LIN {X 0,Y 208.481,Z 945.094,A -85,B 0,C 180,E1 25559.989,E2 25559.989} C_VEL
LIN {X 0,Y 208.561,Z 942.719,A -85,B 0,C 180,E1 25564.152,E2 25564.152} C_VEL
LIN {X 0,Y 203.616,Z 945.932,A -85,B 0,C 180,E1 25571.784,E2 25571.784} C_VEL
LIN {X 0,Y 202.309,Z 947.285,A -85,B 0,C 180,E1 25573.38,E2 25573.38} C_VEL
LIN {X 0,Y 199.131,Z 950.146,A -85,B 0,C 180,E1 25574.216,E2 25574.216} C_VEL
LIN {X 0,Y 170.283,Z 972.979,A -85,B 0,C 180,E1 25579.15,E2 25579.15} C_VEL
LIN {X 0,Y 139.935,Z 991.586,A -85,B 0,C 180,E1 25586.801,E2 25586.801} C_VEL
LIN {X 0,Y 111.609,Z 1004.959,A -85,B 0,C 180,E1 25598.741,E2 25598.741} C_VEL
LIN {X 0,Y 89.534,Z 1013.124,A -85,B 0,C 180,E1 25617.669,E2 25617.669} C_VEL
LIN {X 0,Y 80.233,Z 1016.11,A -85,B 0,C 180,E1 25639.124,E2 25639.124} C_VEL
LIN {X 0,Y 80.25,Z 1016.086,A -85,B 0,C 180,E1 25660.875,E2 25660.875} C_VEL
LIN {X 0,Y 95.67,Z 1010.987,A -85,B 0,C 180,E1 25689.273,E2 25689.273} C_VEL
LIN {X 0,Y 122.761,Z 1000.055,A -85,B 0,C 180,E1 25706.77,E2 25706.77} C_VEL
LIN {X 0,Y 152.69,Z 984.282,A -85,B 0,C 180,E1 25716.747,E2 25716.747} C_VEL
LIN {X 0,Y 184.293,Z 962.437,A -85,B 0,C 180,E1 25723.376,E2 25723.376} C_VEL
LIN {X 0,Y 191.521,Z 956.574,A -85,B 0,C 180,E1 25724.562,E2 25724.562} C_VEL
LIN {X 0,Y 196.197,Z 952.595,A -85,B 0,C 180,E1 25726.225,E2 25726.225} C_VEL
LIN {X 0,Y 199.352,Z 949.805,A -85,B 0,C 180,E1 25729.978,E2 25729.978} C_VEL
LIN {X 0,Y 201.389,Z 948.643,A -85,B 0,C 180,E1 25734.136,E2 25734.136} C_VEL
LIN {X 0,Y 202.552,Z 948.131,A -85,B 0,C 180,E1 25735.725,E2 25735.725} C_VEL
LIN {X 0,Y 202.66,Z 949.809,A -85,B 0,C 180,E1 25739.218,E2 25739.218} C_VEL
LIN {X 0,Y 170.919,Z 977.867,A -85,B 0,C 180,E1 25743.237,E2 25743.237} C_VEL
LIN {X 0,Y 136.439,Z 1002.048,A -85,B 0,C 180,E1 25749.996,E2 25749.996} C_VEL
LIN {X 0,Y 103.347,Z 1020.966,A -85,B 0,C 180,E1 25762.119,E2 25762.119} C_VEL
LIN {X 0,Y 78.07,Z 1033.952,A -85,B 0,C 180,E1 25783.511,E2 25783.511} C_VEL
LIN {X 0,Y 69.524,Z 1039.389,A -85,B 0,C 180,E1 25804.18,E2 25804.18} C_VEL
LIN {X 0,Y 69.25,Z 1042.157,A -85,B 0,C 180,E1 25829.999,E2 25829.999} C_VEL
LIN {X 0,Y 69.527,Z 1039.414,A -85,B 0,C 180,E1 25855.817,E2 25855.817} C_VEL
LIN {X 0,Y 84.225,Z 1030.826,A -85,B 0,C 180,E1 25883.987,E2 25883.987} C_VEL
LIN {X 0,Y 114.045,Z 1015.315,A -85,B 0,C 180,E1 25902.786,E2 25902.786} C_VEL
LIN {X 0,Y 148.793,Z 994.172,A -85,B 0,C 180,E1 25912.78,E2 25912.78} C_VEL
LIN {X 0,Y 181.759,Z 969.208,A -85,B 0,C 180,E1 25918.286,E2 25918.286} C_VEL
LIN {X 0,Y 202.744,Z 949.964,A -85,B 0,C 180,E1 25920.772,E2 25920.772} C_VEL
LIN {X 0,Y 202.608,Z 948.314,A -85,B 0,C 180,E1 25924.274,E2 25924.274} C_VEL
LIN {X 0,Y 198.102,Z 950.964,A -85,B 0,C 180,E1 25931,E2 25931} C_VEL
LIN {X 0,Y 196.097,Z 952.662,A -85,B 0,C 180,E1 25932.195,E2 25932.195} C_VEL
LIN {X 0,Y 166.195,Z 975.484,A -85,B 0,C 180,E1 25936.959,E2 25936.959} C_VEL
LIN {X 0,Y 136.428,Z 993.025,A -85,B 0,C 180,E1 25943.915,E2 25943.915} C_VEL
LIN {X 0,Y 106.882,Z 1006.314,A -85,B 0,C 180,E1 25955.464,E2 25955.464} C_VEL
LIN {X 0,Y 85.596,Z 1013.77,A -85,B 0,C 180,E1 25971.753,E2 25971.753} C_VEL
LIN {X 0,Y 72.588,Z 1017.461,A -85,B 0,C 180,E1 25997.962,E2 25997.962} C_VEL
LIN {X 0,Y 71.763,Z 1017.732,A -85,B 0,C 180,E1 26010.001,E2 26010.001} C_VEL
LIN {X 0,Y 76.046,Z 1016.46,A -85,B 0,C 180,E1 26033.465,E2 26033.465} C_VEL
LIN {X 0,Y 94.294,Z 1010.865,A -85,B 0,C 180,E1 26056.264,E2 26056.264} C_VEL
LIN {X 0,Y 121.226,Z 1000.274,A -85,B 0,C 180,E1 26070.955,E2 26070.955} C_VEL
LIN {X 0,Y 152.847,Z 983.799,A -85,B 0,C 180,E1 26080.221,E2 26080.221} C_VEL
LIN {X 0,Y 184.689,Z 961.877,A -85,B 0,C 180,E1 26086.112,E2 26086.112} C_VEL
LIN {X 0,Y 196.094,Z 952.434,A -85,B 0,C 180,E1 26087.749,E2 26087.749} C_VEL
LIN {X 0,Y 198.088,Z 950.746,A -85,B 0,C 180,E1 26088.999,E2 26088.999} C_VEL
LIN {X 0,Y 201.389,Z 948.643,A -85,B 0,C 180,E1 26094.136,E2 26094.136} C_VEL
LIN {X 0,Y 200.229,Z 950.371,A -85,B 0,C 180,E1 26095.822,E2 26095.822} C_VEL
LIN {X 0,Y 195.34,Z 955.454,A -85,B 0,C 180,E1 26097.311,E2 26097.311} C_VEL
LIN {X 0,Y 188.146,Z 962.065,A -85,B 0,C 180,E1 26098.362,E2 26098.362} C_VEL
LIN {X 0,Y 153.922,Z 988.562,A -85,B 0,C 180,E1 26102.846,E2 26102.846} C_VEL
LIN {X 0,Y 118.999,Z 1009.936,A -85,B 0,C 180,E1 26110.728,E2 26110.728} C_VEL
LIN {X 0,Y 87.096,Z 1025.846,A -85,B 0,C 180,E1 26125.16,E2 26125.16} C_VEL
LIN {X 0,Y 67.103,Z 1035.132,A -85,B 0,C 180,E1 26147.399,E2 26147.399} C_VEL
LIN {X 0,Y 60.349,Z 1039.863,A -85,B 0,C 180,E1 26175.47,E2 26175.47} C_VEL
LIN {X 0,Y 61.337,Z 1040.787,A -85,B 0,C 180,E1 26189.999,E2 26189.999} C_VEL
LIN {X 0,Y 62.268,Z 1037.997,A -85,B 0,C 180,E1 26219.095,E2 26219.095} C_VEL
LIN {X 0,Y 79.564,Z 1029.365,A -85,B 0,C 180,E1 26248.901,E2 26248.901} C_VEL
LIN {X 0,Y 111.658,Z 1013.924,A -85,B 0,C 180,E1 26266.888,E2 26266.888} C_VEL
LIN {X 0,Y 146.132,Z 993.898,A -85,B 0,C 180,E1 26275.699,E2 26275.699} C_VEL
LIN {X 0,Y 179.53,Z 969.516,A -85,B 0,C 180,E1 26280.687,E2 26280.687} C_VEL
LIN {X 0,Y 197.003,Z 954.289,A -85,B 0,C 180,E1 26282.488,E2 26282.488} C_VEL
LIN {X 0,Y 196.533,Z 953.833,A -85,B 0,C 180,E1 26284.406,E2 26284.406} C_VEL
LIN {X 0,Y 192.985,Z 955.536,A -85,B 0,C 180,E1 26289.494,E2 26289.494} C_VEL
LIN {X 0,Y 191.197,Z 956.979,A -85,B 0,C 180,E1 26290.4,E2 26290.4} C_VEL
LIN {X 0,Y 158.897,Z 980.258,A -85,B 0,C 180,E1 26295.266,E2 26295.266} C_VEL
LIN {X 0,Y 127.117,Z 997.521,A -85,B 0,C 180,E1 26302.626,E2 26302.626} C_VEL
LIN {X 0,Y 94.244,Z 1010.583,A -85,B 0,C 180,E1 26316.562,E2 26316.562} C_VEL
LIN {X 0,Y 74.594,Z 1016.422,A -85,B 0,C 180,E1 26334.219,E2 26334.219} C_VEL
LIN {X 0,Y 63.996,Z 1019.077,A -85,B 0,C 180,E1 26370.001,E2 26370.001} C_VEL
LIN {X 0,Y 74.98,Z 1016.276,A -85,B 0,C 180,E1 26406.188,E2 26406.188} C_VEL
LIN {X 0,Y 99.778,Z 1008.6,A -85,B 0,C 180,E1 26426.569,E2 26426.569} C_VEL
LIN {X 0,Y 130.415,Z 995.771,A -85,B 0,C 180,E1 26438.238,E2 26438.238} C_VEL
LIN {X 0,Y 162.406,Z 977.795,A -85,B 0,C 180,E1 26445.282,E2 26445.282} C_VEL
LIN {X 0,Y 191.22,Z 956.727,A -85,B 0,C 180,E1 26449.567,E2 26449.567} C_VEL
LIN {X 0,Y 193.337,Z 955.08,A -85,B 0,C 180,E1 26451.002,E2 26451.002} C_VEL
LIN {X 0,Y 196.513,Z 953.635,A -85,B 0,C 180,E1 26455.593,E2 26455.593} C_VEL
LIN {X 0,Y 196.99,Z 953.973,A -85,B 0,C 180,E1 26457.275,E2 26457.275} C_VEL
LIN {X 0,Y 188.146,Z 962.065,A -85,B 0,C 180,E1 26458.362,E2 26458.362} C_VEL
LIN {X 0,Y 174.299,Z 972.838,A -85,B 0,C 180,E1 26458.579,E2 26458.579} C_VEL
LIN {X 0,Y 159.892,Z 982.792,A -85,B 0,C 180,E1 26458.877,E2 26458.877} C_VEL
LIN {X 0,Y 124.729,Z 1004.643,A -85,B 0,C 180,E1 26464.941,E2 26464.941} C_VEL
LIN {X 0,Y 90.673,Z 1021.379,A -85,B 0,C 180,E1 26476.238,E2 26476.238} C_VEL
LIN {X 0,Y 63.969,Z 1032.548,A -85,B 0,C 180,E1 26497.857,E2 26497.857} C_VEL
LIN {X 0,Y 55.242,Z 1036.551,A -85,B 0,C 180,E1 26516.76,E2 26516.76} C_VEL
LIN {X 0,Y 53.421,Z 1039.416,A -85,B 0,C 180,E1 26549.999,E2 26549.999} C_VEL
LIN {X 0,Y 55.996,Z 1036.167,A -85,B 0,C 180,E1 26585.732,E2 26585.732} C_VEL
LIN {X 0,Y 77.603,Z 1027.018,A -85,B 0,C 180,E1 26615.958,E2 26615.958} C_VEL
LIN {X 0,Y 110.855,Z 1012.045,A -85,B 0,C 180,E1 26631.405,E2 26631.405} C_VEL
LIN {X 0,Y 147.623,Z 991.18,A -85,B 0,C 180,E1 26639.34,E2 26639.34} C_VEL
LIN {X 0,Y 182.03,Z 966.196,A -85,B 0,C 180,E1 26643.568,E2 26643.568} C_VEL
LIN {X 0,Y 190.255,Z 959.17,A -85,B 0,C 180,E1 26644.552,E2 26644.552} C_VEL
LIN {X 0,Y 188.055,Z 960.104,A -85,B 0,C 180,E1 26647.598,E2 26647.598} C_VEL
LIN {X 0,Y 186.21,Z 961.356,A -85,B 0,C 180,E1 26648.52,E2 26648.52} C_VEL
LIN {X 0,Y 153.497,Z 983.679,A -85,B 0,C 180,E1 26653.094,E2 26653.094} C_VEL
LIN {X 0,Y 120.978,Z 1000.302,A -85,B 0,C 180,E1 26660.185,E2 26660.185} C_VEL
LIN {X 0,Y 89.81,Z 1011.934,A -85,B 0,C 180,E1 26672.555,E2 26672.555} C_VEL
LIN {X 0,Y 69.429,Z 1017.52,A -85,B 0,C 180,E1 26689.143,E2 26689.143} C_VEL
LIN {X 0,Y 57.436,Z 1020.161,A -85,B 0,C 180,E1 26714.717,E2 26714.717} C_VEL
LIN {X 0,Y 56.215,Z 1020.425,A -85,B 0,C 180,E1 26730.001,E2 26730.001} C_VEL
LIN {X 0,Y 62.04,Z 1019.166,A -85,B 0,C 180,E1 26759.215,E2 26759.215} C_VEL
LIN {X 0,Y 84.258,Z 1013.575,A -85,B 0,C 180,E1 26783.959,E2 26783.959} C_VEL
LIN {X 0,Y 114.463,Z 1002.997,A -85,B 0,C 180,E1 26797.804,E2 26797.804} C_VEL
LIN {X 0,Y 148.299,Z 986.544,A -85,B 0,C 180,E1 26805.898,E2 26805.898} C_VEL
LIN {X 0,Y 181.094,Z 965.062,A -85,B 0,C 180,E1 26810.817,E2 26810.817} C_VEL
LIN {X 0,Y 186.185,Z 961.16,A -85,B 0,C 180,E1 26811.424,E2 26811.424} C_VEL
LIN {X 0,Y 188.053,Z 959.89,A -85,B 0,C 180,E1 26812.363,E2 26812.363} C_VEL
LIN {X 0,Y 190.247,Z 958.961,A -85,B 0,C 180,E1 26815.448,E2 26815.448} C_VEL
LIN {X 0,Y 159.892,Z 982.792,A -85,B 0,C 180,E1 26818.877,E2 26818.877} C_VEL
LIN {X 0,Y 144.954,Z 992.033,A -85,B 0,C 180,E1 26819.311,E2 26819.311} C_VEL
LIN {X 0,Y 129.62,Z 1000.319,A -85,B 0,C 180,E1 26820.051,E2 26820.051} C_VEL
LIN {X 0,Y 92.14,Z 1018.502,A -85,B 0,C 180,E1 26829.635,E2 26829.635} C_VEL
LIN {X 0,Y 60.304,Z 1030.74,A -85,B 0,C 180,E1 26850.181,E2 26850.181} C_VEL
LIN {X 0,Y 48.583,Z 1035.127,A -85,B 0,C 180,E1 26871.443,E2 26871.443} C_VEL
LIN {X 0,Y 45.456,Z 1038.036,A -85,B 0,C 180,E1 26910.215,E2 26910.215} C_VEL
LIN {X 0,Y 48.588,Z 1035.156,A -85,B 0,C 180,E1 26948.548,E2 26948.548} C_VEL
LIN {X 0,Y 74.079,Z 1025.748,A -85,B 0,C 180,E1 26981.571,E2 26981.571} C_VEL
LIN {X 0,Y 109.912,Z 1010.576,A -85,B 0,C 180,E1 26995.753,E2 26995.753} C_VEL
LIN {X 0,Y 147.708,Z 989.735,A -85,B 0,C 180,E1 27002.61,E2 27002.61} C_VEL
LIN {X 0,Y 181.435,Z 965.747,A -85,B 0,C 180,E1 27006.083,E2 27006.083} C_VEL
LIN {X 0,Y 178.5,Z 967.827,A -85,B 0,C 180,E1 27006.865,E2 27006.865} C_VEL
LIN {X 0,Y 142.994,Z 990.031,A -85,B 0,C 180,E1 27011.661,E2 27011.661} C_VEL
LIN {X 0,Y 108.313,Z 1005.767,A -85,B 0,C 180,E1 27019.352,E2 27019.352} C_VEL
LIN {X 0,Y 74.136,Z 1016.459,A -85,B 0,C 180,E1 27035.229,E2 27035.229} C_VEL
LIN {X 0,Y 55.339,Z 1020.551,A -85,B 0,C 180,E1 27056.829,E2 27056.829} C_VEL
LIN {X 0,Y 48.447,Z 1021.771,A -85,B 0,C 180,E1 27090.001,E2 27090.001} C_VEL
LIN {X 0,Y 60.401,Z 1019.589,A -85,B 0,C 180,E1 27131.301,E2 27131.301} C_VEL
LIN {X 0,Y 92.087,Z 1011.312,A -85,B 0,C 180,E1 27154.723,E2 27154.723} C_VEL
LIN {X 0,Y 125.467,Z 998.495,A -85,B 0,C 180,E1 27164.874,E2 27164.874} C_VEL
LIN {X 0,Y 159.161,Z 980.563,A -85,B 0,C 180,E1 27170.719,E2 27170.719} C_VEL
LIN {X 0,Y 178.711,Z 967.456,A -85,B 0,C 180,E1 27173.117,E2 27173.117} C_VEL
LIN {X 0,Y 181.498,Z 965.489,A -85,B 0,C 180,E1 27173.885,E2 27173.885} C_VEL
LIN {X 0,Y 145.617,Z 990.907,A -85,B 0,C 180,E1 27177.625,E2 27177.625} C_VEL
LIN {X 0,Y 129.62,Z 1000.319,A -85,B 0,C 180,E1 27180.051,E2 27180.051} C_VEL
LIN {X 0,Y 113.806,Z 1007.736,A -85,B 0,C 180,E1 27181.081,E2 27181.081} C_VEL
LIN {X 0,Y 97.76,Z 1014.25,A -85,B 0,C 180,E1 27182.495,E2 27182.495} C_VEL
LIN {X 0,Y 63.393,Z 1027.055,A -85,B 0,C 180,E1 27197.191,E2 27197.191} C_VEL
LIN {X 0,Y 41.606,Z 1034.004,A -85,B 0,C 180,E1 27226.775,E2 27226.775} C_VEL
LIN {X 0,Y 37.539,Z 1036.664,A -85,B 0,C 180,E1 27269.998,E2 27269.998} C_VEL
LIN {X 0,Y 42.435,Z 1033.724,A -85,B 0,C 180,E1 27315.523,E2 27315.523} C_VEL
LIN {X 0,Y 71.4,Z 1024.45,A -85,B 0,C 180,E1 27347.727,E2 27347.727} C_VEL
LIN {X 0,Y 111.203,Z 1008.342,A -85,B 0,C 180,E1 27360.515,E2 27360.515} C_VEL
LIN {X 0,Y 149.532,Z 987.498,A -85,B 0,C 180,E1 27366.022,E2 27366.022} C_VEL
LIN {X 0,Y 155.275,Z 983.914,A -85,B 0,C 180,E1 27366.579,E2 27366.579} C_VEL
LIN {X 0,Y 120.064,Z 1001.594,A -85,B 0,C 180,E1 27372.245,E2 27372.245} C_VEL
LIN {X 0,Y 88.554,Z 1012.908,A -85,B 0,C 180,E1 27380.805,E2 27380.805} C_VEL
LIN {X 0,Y 58.517,Z 1020.225,A -85,B 0,C 180,E1 27399.089,E2 27399.089} C_VEL
LIN {X 0,Y 42.597,Z 1022.861,A -85,B 0,C 180,E1 27429.182,E2 27429.182} C_VEL
LIN {X 0,Y 40.666,Z 1023.118,A -85,B 0,C 180,E1 27450.001,E2 27450.001} C_VEL
LIN {X 0,Y 49.031,Z 1021.864,A -85,B 0,C 180,E1 27488.14,E2 27488.14} C_VEL
LIN {X 0,Y 76.12,Z 1016.285,A -85,B 0,C 180,E1 27513.514,E2 27513.514} C_VEL
LIN {X 0,Y 109.521,Z 1005.72,A -85,B 0,C 180,E1 27525.392,E2 27525.392} C_VEL
LIN {X 0,Y 145.149,Z 989.377,A -85,B 0,C 180,E1 27531.858,E2 27531.858} C_VEL
LIN {X 0,Y 155.572,Z 983.551,A -85,B 0,C 180,E1 27533.371,E2 27533.371} C_VEL
LIN {X 0,Y 117.838,Z 1005.099,A -85,B 0,C 180,E1 27538.229,E2 27538.229} C_VEL
LIN {X 0,Y 97.76,Z 1014.25,A -85,B 0,C 180,E1 27542.495,E2 27542.495} C_VEL
LIN {X 0,Y 81.484,Z 1019.912,A -85,B 0,C 180,E1 27544.592,E2 27544.592} C_VEL
LIN {X 0,Y 65.026,Z 1024.534,A -85,B 0,C 180,E1 27547.795,E2 27547.795} C_VEL
LIN {X 0,Y 37.104,Z 1032.259,A -85,B 0,C 180,E1 27575.303,E2 27575.303} C_VEL
LIN {X 0,Y 29.543,Z 1035.28,A -85,B 0,C 180,E1 27629.998,E2 27629.998} C_VEL
LIN {X 0,Y 37.104,Z 1032.288,A -85,B 0,C 180,E1 27684.692,E2 27684.692} C_VEL
LIN {X 0,Y 70.091,Z 1022.984,A -85,B 0,C 180,E1 27714.495,E2 27714.495} C_VEL
LIN {X 0,Y 111.495,Z 1006.919,A -85,B 0,C 180,E1 27724.858,E2 27724.858} C_VEL
LIN {X 0,Y 126.179,Z 999.786,A -85,B 0,C 180,E1 27726.873,E2 27726.873} C_VEL
LIN {X 0,Y 111.394,Z 1005.798,A -85,B 0,C 180,E1 27729.817,E2 27729.817} C_VEL
LIN {X 0,Y 79.67,Z 1016.006,A -85,B 0,C 180,E1 27738.168,E2 27738.168} C_VEL
LIN {X 0,Y 46.159,Z 1022.815,A -85,B 0,C 180,E1 27760.926,E2 27760.926} C_VEL
LIN {X 0,Y 32.897,Z 1024.464,A -85,B 0,C 180,E1 27810.002,E2 27810.002} C_VEL
LIN {X 0,Y 46.448,Z 1022.741,A -85,B 0,C 180,E1 27859.383,E2 27859.383} C_VEL
LIN {X 0,Y 79.703,Z 1015.923,A -85,B 0,C 180,E1 27881.765,E2 27881.765} C_VEL
LIN {X 0,Y 118.679,Z 1002.82,A -85,B 0,C 180,E1 27891.37,E2 27891.37} C_VEL
LIN {X 0,Y 126.095,Z 999.712,A -85,B 0,C 180,E1 27893.123,E2 27893.123} C_VEL
LIN {X 0,Y 86.928,Z 1017.032,A -85,B 0,C 180,E1 27900.026,E2 27900.026} C_VEL
LIN {X 0,Y 65.026,Z 1024.534,A -85,B 0,C 180,E1 27907.795,E2 27907.795} C_VEL
LIN {X 0,Y 48.765,Z 1028.181,A -85,B 0,C 180,E1 27913.264,E2 27913.264} C_VEL
LIN {X 0,Y 32.912,Z 1030.836,A -85,B 0,C 180,E1 27923.579,E2 27923.579} C_VEL
LIN {X 0,Y 21.549,Z 1033.895,A -85,B 0,C 180,E1 27989.997,E2 27989.997} C_VEL
LIN {X 0,Y 33.003,Z 1030.848,A -85,B 0,C 180,E1 28056.558,E2 28056.558} C_VEL
LIN {X 0,Y 70.1,Z 1021.426,A -85,B 0,C 180,E1 28081.494,E2 28081.494} C_VEL
LIN {X 0,Y 97.391,Z 1011.851,A -85,B 0,C 180,E1 28087.202,E2 28087.202} C_VEL
LIN {X 0,Y 82.822,Z 1016.043,A -85,B 0,C 180,E1 28091.179,E2 28091.179} C_VEL
LIN {X 0,Y 50.158,Z 1022.93,A -85,B 0,C 180,E1 28105.109,E2 28105.109} C_VEL
LIN {X 0,Y 28.568,Z 1025.562,A -85,B 0,C 180,E1 28138,E2 28138} C_VEL
LIN {X 0,Y 25.103,Z 1025.814,A -85,B 0,C 180,E1 28170.002,E2 28170.002} C_VEL
LIN {X 0,Y 37.994,Z 1024.57,A -85,B 0,C 180,E1 28222.843,E2 28222.843} C_VEL
LIN {X 0,Y 70.542,Z 1019.003,A -85,B 0,C 180,E1 28244.974,E2 28244.974} C_VEL
LIN {X 0,Y 92.006,Z 1013.302,A -85,B 0,C 180,E1 28250.872,E2 28250.872} C_VEL
LIN {X 0,Y 97.531,Z 1011.701,A -85,B 0,C 180,E1 28252.757,E2 28252.757} C_VEL
LIN {X 0,Y 56.874,Z 1025.178,A -85,B 0,C 180,E1 28263.362,E2 28263.362} C_VEL
LIN {X 0,Y 32.912,Z 1030.836,A -85,B 0,C 180,E1 28283.579,E2 28283.579} C_VEL
LIN {X 0,Y 22.965,Z 1032.258,A -85,B 0,C 180,E1 28301.464,E2 28301.464} C_VEL
LIN {X 0,Y 14.696,Z 1032.569,A -85,B 0,C 180,E1 28334.454,E2 28334.454} C_VEL
LIN {X 0,Y 13.198,Z 1032.165,A -85,B 0,C 180,E1 28371.239,E2 28371.239} C_VEL
LIN {X 0,Y 36.928,Z 1028.247,A -85,B 0,C 180,E1 28436.174,E2 28436.174} C_VEL
LIN {X 0,Y 69.266,Z 1020.44,A -85,B 0,C 180,E1 28448.058,E2 28448.058} C_VEL
LIN {X 0,Y 47.373,Z 1024.284,A -85,B 0,C 180,E1 28456.516,E2 28456.516} C_VEL
LIN {X 0,Y 22.35,Z 1026.91,A -85,B 0,C 180,E1 28487.362,E2 28487.362} C_VEL
LIN {X 0,Y 17.333,Z 1027.16,A -85,B 0,C 180,E1 28530.004,E2 28530.004} C_VEL
LIN {X 0,Y 34.174,Z 1025.888,A -85,B 0,C 180,E1 28593.779,E2 28593.779} C_VEL
LIN {X 0,Y 61.66,Z 1021.808,A -85,B 0,C 180,E1 28609.166,E2 28609.166} C_VEL
LIN {X 0,Y 69.284,Z 1020.373,A -85,B 0,C 180,E1 28611.942,E2 28611.942} C_VEL
LIN {X 0,Y 28.124,Z 1029.799,A -85,B 0,C 180,E1 28631.81,E2 28631.81} C_VEL
LIN {X 0,Y 13.522,Z 1032.505,A -85,B 0,C 180,E1 28709.995,E2 28709.995} C_VEL
LIN {X 0,Y 13.198,Z 1032.165,A -85,B 0,C 180,E1 28731.239,E2 28731.239} C_VEL
LIN {X 0,Y 17.713,Z 1030.8,A -85,B 0,C 180,E1 28778.396,E2 28778.396} C_VEL
LIN {X 0,Y 35.288,Z 1027.148,A -85,B 0,C 180,E1 28808.439,E2 28808.439} C_VEL
LIN {X 0,Y 31.153,Z 1027.306,A -85,B 0,C 180,E1 28813.603,E2 28813.603} C_VEL
LIN {X 0,Y 9.538,Z 1028.51,A -85,B 0,C 180,E1 28890.006,E2 28890.006} C_VEL
LIN {X 0,Y 31.16,Z 1027.274,A -85,B 0,C 180,E1 28966.357,E2 28966.357} C_VEL
LIN {X 0,Y 35.96,Z 1027.005,A -85,B 0,C 180,E1 28971.339,E2 28971.339} C_VEL
LIN {X 0,Y 15.213,Z 1029.998,A -85,B 0,C 180,E1 28985.589,E2 28985.589} C_VEL
LIN {X 0,Y 5.49,Z 1031.113,A -85,B 0,C 180,E1 29069.989,E2 29069.989} C_VEL
LIN {X 0,Y 30.478,Z 1027.973,A -85,B 0,C 180,E1 29166.556,E2 29166.556} C_VEL
LIN {X 0,Y 35.288,Z 1027.148,A -85,B 0,C 180,E1 29168.439,E2 29168.439} C_VEL
LIN {X 0,Y 37.572,Z 1029.121,A -85,B 0,C 180,E1 29169.161,E2 29169.161} C_VEL
LIN {X 0,Y 37.572,Z 1104,A -85,B 0,C 180,E1 29169.161,E2 29169.161} C_VEL
LIN {X 0,Y 37.572,Z 1104,A -85,B 0,C 180,E1 29169.161,E2 29169.161}

QRS_NEXT_CUT()
PTP {E1 29337.043,E2 29337.043}
PTP {X 0,Y 607.835,A -85,B 0,C 180,E1 29337.043,E2 29337.043,E3 0,E4 0,E5 0,E6 0}
QRS_SPEED_INIT()
LIN {X 0,Y 607.835,Z 1104,A -85,B 0,C 180,E1 29337.043,E2 29337.043,E3 0,E4 0,E5 0,E6 0} C_VEL
LIN {X 0,Y 607.835,Z 381.402,A -85,B 0,C 180,E1 29337.043,E2 29337.043} C_VEL
LIN {X 0,Y 607.835,Z 373.326,A -85,B 0,C 180,E1 29337.043,E2 29337.043} C_VEL
LIN {X 0,Y 607.835,Z 371.326,A -85,B 0,C 180,E1 29336.855,E2 29336.855} C_VEL
LIN {X 0,Y 607.918,Z 371.324,A -85,B 0,C 180,E1 29333.768,E2 29333.768} C_VEL
LIN {X 0,Y 607.836,Z 371.325,A -85,B 0,C 180,E1 29330.723,E2 29330.723} C_VEL
LIN {X 0,Y 607.886,Z 371.327,A -85,B 0,C 180,E1 29327.846,E2 29327.846} C_VEL
LIN {X 0,Y 607.847,Z 371.324,A -85,B 0,C 180,E1 29324.74,E2 29324.74} C_VEL
LIN {X 0,Y 607.849,Z 371.326,A -85,B 0,C 180,E1 29321.946,E2 29321.946} C_VEL
LIN {X 0,Y 607.866,Z 371.324,A -85,B 0,C 180,E1 29318.683,E2 29318.683} C_VEL
LIN {X 0,Y 607.838,Z 371.326,A -85,B 0,C 180,E1 29315.916,E2 29315.916} C_VEL
LIN {X 0,Y 607.919,Z 371.324,A -85,B 0,C 180,E1 29312.849,E2 29312.849} C_VEL
LIN {X 0,Y 607.839,Z 371.324,A -85,B 0,C 180,E1 29309.778,E2 29309.778} C_VEL
LIN {X 0,Y 607.908,Z 371.328,A -85,B 0,C 180,E1 29306.79,E2 29306.79} C_VEL
LIN {X 0,Y 607.844,Z 371.323,A -85,B 0,C 180,E1 29303.688,E2 29303.688} C_VEL
LIN {X 0,Y 607.871,Z 371.327,A -85,B 0,C 180,E1 29300.83,E2 29300.83} C_VEL
LIN {X 0,Y 607.854,Z 371.324,A -85,B 0,C 180,E1 29297.591,E2 29297.591} C_VEL
LIN {X 0,Y 607.848,Z 371.325,A -85,B 0,C 180,E1 29294.849,E2 29294.849} C_VEL
LIN {X 0,Y 607.894,Z 371.322,A -85,B 0,C 180,E1 29291.691,E2 29291.691} C_VEL
LIN {X 0,Y 607.843,Z 371.326,A -85,B 0,C 180,E1 29288.767,E2 29288.767} C_VEL
LIN {X 0,Y 607.917,Z 371.325,A -85,B 0,C 180,E1 29285.724,E2 29285.724} C_VEL
LIN {X 0,Y 607.889,Z 371.537,A -85,B 0,C 180,E1 29283.975,E2 29283.975} C_VEL
LIN {X 0,Y 607.908,Z 373.819,A -85,B 0,C 180,E1 29283.775,E2 29283.775} C_VEL
LIN {X 0,Y 607.876,Z 417.731,A -85,B 0,C 180,E1 29280.932,E2 29280.932} C_VEL
LIN {X 0,Y 607.895,Z 463.368,A -85,B 0,C 180,E1 29278.061,E2 29278.061} C_VEL
LIN {X 0,Y 607.889,Z 470.207,A -85,B 0,C 180,E1 29277.648,E2 29277.648} C_VEL
LIN {X 0,Y 607.906,Z 714.954,A -85,B 0,C 180,E1 29274.487,E2 29274.487} C_VEL
LIN {X 0,Y 607.916,Z 737.553,A -85,B 0,C 180,E1 29274.138,E2 29274.138} C_VEL
LIN {X 0,Y 607.905,Z 756.795,A -85,B 0,C 180,E1 29273.687,E2 29273.687} C_VEL
LIN {X 0,Y 607.915,Z 776.617,A -85,B 0,C 180,E1 29273.045,E2 29273.045} C_VEL
LIN {X 0,Y 607.906,Z 794.968,A -85,B 0,C 180,E1 29272.279,E2 29272.279} C_VEL
LIN {X 0,Y 607.918,Z 813.819,A -85,B 0,C 180,E1 29271.315,E2 29271.315} C_VEL
LIN {X 0,Y 607.917,Z 831.797,A -85,B 0,C 180,E1 29270.206,E2 29270.206} C_VEL
LIN {X 0,Y 607.916,Z 848.757,A -85,B 0,C 180,E1 29268.964,E2 29268.964} C_VEL
LIN {X 0,Y 607.916,Z 864.943,A -85,B 0,C 180,E1 29267.566,E2 29267.566} C_VEL
LIN {X 0,Y 607.909,Z 879.945,A -85,B 0,C 180,E1 29266.041,E2 29266.041} C_VEL
LIN {X 0,Y 607.915,Z 893.927,A -85,B 0,C 180,E1 29264.361,E2 29264.361} C_VEL
LIN {X 0,Y 607.917,Z 905.994,A -85,B 0,C 180,E1 29262.636,E2 29262.636} C_VEL
LIN {X 0,Y 607.907,Z 916.116,A -85,B 0,C 180,E1 29260.903,E2 29260.903} C_VEL
LIN {X 0,Y 607.901,Z 924.868,A -85,B 0,C 180,E1 29259.085,E2 29259.085} C_VEL
LIN {X 0,Y 607.9,Z 931.847,A -85,B 0,C 180,E1 29257.276,E2 29257.276} C_VEL
LIN {X 0,Y 607.901,Z 937.387,A -85,B 0,C 180,E1 29255.38,E2 29255.38} C_VEL
LIN {X 0,Y 607.9,Z 941.164,A -85,B 0,C 180,E1 29253.489,E2 29253.489} C_VEL
LIN {X 0,Y 607.903,Z 943.341,A -85,B 0,C 180,E1 29251.602,E2 29251.602} C_VEL
LIN {X 0,Y 607.904,Z 943.95,A -85,B 0,C 180,E1 29249.717,E2 29249.717} C_VEL
LIN {X 0,Y 607.915,Z 942.998,A -85,B 0,C 180,E1 29247.832,E2 29247.832} C_VEL
LIN {X 0,Y 607.917,Z 940.209,A -85,B 0,C 180,E1 29245.85,E2 29245.85} C_VEL
LIN {X 0,Y 607.915,Z 935.855,A -85,B 0,C 180,E1 29243.958,E2 29243.958} C_VEL
LIN {X 0,Y 607.91,Z 929.786,A -85,B 0,C 180,E1 29242.059,E2 29242.059} C_VEL
LIN {X 0,Y 607.905,Z 922.315,A -85,B 0,C 180,E1 29240.246,E2 29240.246} C_VEL
LIN {X 0,Y 607.904,Z 912.972,A -85,B 0,C 180,E1 29238.424,E2 29238.424} C_VEL
LIN {X 0,Y 607.906,Z 902.111,A -85,B 0,C 180,E1 29236.687,E2 29236.687} C_VEL
LIN {X 0,Y 607.914,Z 889.841,A -85,B 0,C 180,E1 29235.035,E2 29235.035} C_VEL
LIN {X 0,Y 607.917,Z 876.164,A -85,B 0,C 180,E1 29233.469,E2 29233.469} C_VEL
LIN {X 0,Y 607.912,Z 861,A -85,B 0,C 180,E1 29231.988,E2 29231.988} C_VEL
LIN {X 0,Y 607.918,Z 844.197,A -85,B 0,C 180,E1 29230.595,E2 29230.595} C_VEL
LIN {X 0,Y 607.917,Z 827.063,A -85,B 0,C 180,E1 29229.392,E2 29229.392} C_VEL
LIN {X 0,Y 607.918,Z 808.945,A -85,B 0,C 180,E1 29228.322,E2 29228.322} C_VEL
LIN {X 0,Y 607.914,Z 790.231,A -85,B 0,C 180,E1 29227.415,E2 29227.415} C_VEL
LIN {X 0,Y 607.917,Z 771.118,A -85,B 0,C 180,E1 29226.673,E2 29226.673} C_VEL
LIN {X 0,Y 607.906,Z 751.358,A -85,B 0,C 180,E1 29226.082,E2 29226.082} C_VEL
LIN {X 0,Y 607.913,Z 731.468,A -85,B 0,C 180,E1 29225.657,E2 29225.657} C_VEL
LIN {X 0,Y 607.883,Z 470.115,A -85,B 0,C 180,E1 29222.258,E2 29222.258} C_VEL
LIN {X 0,Y 607.878,Z 425.789,A -85,B 0,C 180,E1 29219.491,E2 29219.491} C_VEL
LIN {X 0,Y 607.917,Z 380.359,A -85,B 0,C 180,E1 29216.565,E2 29216.565} C_VEL
LIN {X 0,Y 607.895,Z 371.672,A -85,B 0,C 180,E1 29215.966,E2 29215.966} C_VEL
LIN {X 0,Y 607.851,Z 371.324,A -85,B 0,C 180,E1 29215.31,E2 29215.31} C_VEL
LIN {X 0,Y 607.919,Z 371.321,A -85,B 0,C 180,E1 29212.277,E2 29212.277} C_VEL
LIN {X 0,Y 607.852,Z 371.324,A -85,B 0,C 180,E1 29209.171,E2 29209.171} C_VEL
LIN {X 0,Y 607.9,Z 371.321,A -85,B 0,C 180,E1 29206.175,E2 29206.175} C_VEL
LIN {X 0,Y 607.857,Z 371.325,A -85,B 0,C 180,E1 29203.05,E2 29203.05} C_VEL
LIN {X 0,Y 607.871,Z 371.322,A -85,B 0,C 180,E1 29200.15,E2 29200.15} C_VEL
LIN {X 0,Y 607.864,Z 371.325,A -85,B 0,C 180,E1 29196.897,E2 29196.897} C_VEL
LIN {X 0,Y 607.859,Z 371.323,A -85,B 0,C 180,E1 29194.001,E2 29194.001} C_VEL
LIN {X 0,Y 607.864,Z 371.325,A -85,B 0,C 180,E1 29190.658,E2 29190.658} C_VEL
LIN {X 0,Y 607.85,Z 371.324,A -85,B 0,C 180,E1 29187.85,E2 29187.85} C_VEL
LIN {X 0,Y 607.898,Z 371.327,A -85,B 0,C 180,E1 29184.694,E2 29184.694} C_VEL
LIN {X 0,Y 607.844,Z 371.324,A -85,B 0,C 180,E1 29181.723,E2 29181.723} C_VEL
LIN {X 0,Y 607.914,Z 371.327,A -85,B 0,C 180,E1 29178.607,E2 29178.607} C_VEL
LIN {X 0,Y 607.842,Z 371.325,A -85,B 0,C 180,E1 29175.651,E2 29175.651} C_VEL
LIN {X 0,Y 607.893,Z 371.323,A -85,B 0,C 180,E1 29172.733,E2 29172.733} C_VEL
LIN {X 0,Y 607.846,Z 371.326,A -85,B 0,C 180,E1 29169.564,E2 29169.564} C_VEL
LIN {X 0,Y 607.854,Z 371.324,A -85,B 0,C 180,E1 29166.802,E2 29166.802} C_VEL
LIN {X 0,Y 607.858,Z 371.326,A -85,B 0,C 180,E1 29163.49,E2 29163.49} C_VEL
LIN {X 0,Y 607.841,Z 371.325,A -85,B 0,C 180,E1 29160.754,E2 29160.754} C_VEL
LIN {X 0,Y 607.909,Z 371.327,A -85,B 0,C 180,E1 29157.644,E2 29157.644} C_VEL
LIN {X 0,Y 607.836,Z 371.326,A -85,B 0,C 180,E1 29154.715,E2 29154.715} C_VEL
LIN {X 0,Y 607.896,Z 371.323,A -85,B 0,C 180,E1 29151.773,E2 29151.773} C_VEL
LIN {X 0,Y 607.839,Z 371.325,A -85,B 0,C 180,E1 29148.635,E2 29148.635} C_VEL
LIN {X 0,Y 607.849,Z 371.324,A -85,B 0,C 180,E1 29145.91,E2 29145.91} C_VEL
LIN {X 0,Y 607.85,Z 371.326,A -85,B 0,C 180,E1 29142.565,E2 29142.565} C_VEL
LIN {X 0,Y 607.838,Z 371.324,A -85,B 0,C 180,E1 29139.792,E2 29139.792} C_VEL
LIN {X 0,Y 607.889,Z 371.327,A -85,B 0,C 180,E1 29136.647,E2 29136.647} C_VEL
LIN {X 0,Y 607.831,Z 371.325,A -85,B 0,C 180,E1 29133.737,E2 29133.737} C_VEL
LIN {X 0,Y 607.914,Z 371.327,A -85,B 0,C 180,E1 29130.651,E2 29130.651} C_VEL
LIN {X 0,Y 607.832,Z 371.327,A -85,B 0,C 180,E1 29127.683,E2 29127.683} C_VEL
LIN {X 0,Y 607.847,Z 371.325,A -85,B 0,C 180,E1 29124.965,E2 29124.965} C_VEL
LIN {X 0,Y 607.845,Z 371.326,A -85,B 0,C 180,E1 29121.674,E2 29121.674} C_VEL
LIN {X 0,Y 607.829,Z 371.327,A -85,B 0,C 180,E1 29118.979,E2 29118.979} C_VEL
LIN {X 0,Y 607.91,Z 371.328,A -85,B 0,C 180,E1 29115.915,E2 29115.915} C_VEL
LIN {X 0,Y 607.825,Z 371.319,A -85,B 0,C 180,E1 29112.924,E2 29112.924} C_VEL
LIN {X 0,Y 607.883,Z 371.652,A -85,B 0,C 180,E1 29112.08,E2 29112.08} C_VEL
LIN {X 0,Y 607.904,Z 373.549,A -85,B 0,C 180,E1 29111.935,E2 29111.935} C_VEL
LIN {X 0,Y 607.918,Z 430.557,A -85,B 0,C 180,E1 29109.077,E2 29109.077} C_VEL
LIN {X 0,Y 607.904,Z 466.026,A -85,B 0,C 180,E1 29107.384,E2 29107.384} C_VEL
LIN {X 0,Y 607.915,Z 668.583,A -85,B 0,C 180,E1 29104.485,E2 29104.485} C_VEL
LIN {X 0,Y 607.913,Z 815.111,A -85,B 0,C 180,E1 29102.425,E2 29102.425} C_VEL
LIN {X 0,Y 607.914,Z 837.997,A -85,B 0,C 180,E1 29101.932,E2 29101.932} C_VEL
LIN {X 0,Y 607.918,Z 856.544,A -85,B 0,C 180,E1 29101.394,E2 29101.394} C_VEL
LIN {X 0,Y 607.912,Z 877.921,A -85,B 0,C 180,E1 29100.628,E2 29100.628} C_VEL
LIN {X 0,Y 607.919,Z 898.106,A -85,B 0,C 180,E1 29099.726,E2 29099.726} C_VEL
LIN {X 0,Y 607.916,Z 918.757,A -85,B 0,C 180,E1 29098.649,E2 29098.649} C_VEL
LIN {X 0,Y 607.918,Z 938.559,A -85,B 0,C 180,E1 29097.421,E2 29097.421} C_VEL
LIN {X 0,Y 607.912,Z 957.955,A -85,B 0,C 180,E1 29096.05,E2 29096.05} C_VEL
LIN {X 0,Y 607.91,Z 976.18,A -85,B 0,C 180,E1 29094.558,E2 29094.558} C_VEL
LIN {X 0,Y 607.909,Z 994.595,A -85,B 0,C 180,E1 29092.84,E2 29092.84} C_VEL
LIN {X 0,Y 607.916,Z 1010.874,A -85,B 0,C 180,E1 29091.112,E2 29091.112} C_VEL
LIN {X 0,Y 607.913,Z 1026.064,A -85,B 0,C 180,E1 29089.253,E2 29089.253} C_VEL
LIN {X 0,Y 607.913,Z 1040.516,A -85,B 0,C 180,E1 29087.221,E2 29087.221} C_VEL
LIN {X 0,Y 607.9,Z 1052.034,A -85,B 0,C 180,E1 29085.356,E2 29085.356} C_VEL
LIN {X 0,Y 607.885,Z 1062.754,A -85,B 0,C 180,E1 29083.313,E2 29083.313} C_VEL
LIN {X 0,Y 607.907,Z 1071.374,A -85,B 0,C 180,E1 29081.383,E2 29081.383} C_VEL
LIN {X 0,Y 607.896,Z 1079.037,A -85,B 0,C 180,E1 29079.276,E2 29079.276} C_VEL
LIN {X 0,Y 607.894,Z 1084.335,A -85,B 0,C 180,E1 29077.466,E2 29077.466} C_VEL
LIN {X 0,Y 607.908,Z 1089.161,A -85,B 0,C 180,E1 29075.285,E2 29075.285} C_VEL
LIN {X 0,Y 607.884,Z 1091.953,A -85,B 0,C 180,E1 29073.395,E2 29073.395} C_VEL
LIN {X 0,Y 607.909,Z 1093.716,A -85,B 0,C 180,E1 29071.225,E2 29071.225} C_VEL
LIN {X 0,Y 607.883,Z 1093.828,A -85,B 0,C 180,E1 29069.246,E2 29069.246} C_VEL
LIN {X 0,Y 607.895,Z 1092.63,A -85,B 0,C 180,E1 29067.172,E2 29067.172} C_VEL
LIN {X 0,Y 607.903,Z 1089.797,A -85,B 0,C 180,E1 29065.094,E2 29065.094} C_VEL
LIN {X 0,Y 607.882,Z 1085.597,A -85,B 0,C 180,E1 29063.009,E2 29063.009} C_VEL
LIN {X 0,Y 607.913,Z 1079.647,A -85,B 0,C 180,E1 29060.915,E2 29060.915} C_VEL
LIN {X 0,Y 607.897,Z 1072.187,A -85,B 0,C 180,E1 29058.809,E2 29058.809} C_VEL
LIN {X 0,Y 607.887,Z 1063.218,A -85,B 0,C 180,E1 29056.784,E2 29056.784} C_VEL
LIN {X 0,Y 607.911,Z 1053.18,A -85,B 0,C 180,E1 29054.84,E2 29054.84} C_VEL
LIN {X 0,Y 607.912,Z 1041.043,A -85,B 0,C 180,E1 29052.86,E2 29052.86} C_VEL
LIN {X 0,Y 607.912,Z 1027.214,A -85,B 0,C 180,E1 29050.895,E2 29050.895} C_VEL
LIN {X 0,Y 607.917,Z 1012.578,A -85,B 0,C 180,E1 29049.089,E2 29049.089} C_VEL
LIN {X 0,Y 607.905,Z 996.233,A -85,B 0,C 180,E1 29047.325,E2 29047.325} C_VEL
LIN {X 0,Y 607.905,Z 978.853,A -85,B 0,C 180,E1 29045.67,E2 29045.67} C_VEL
LIN {X 0,Y 607.908,Z 960.603,A -85,B 0,C 180,E1 29044.16,E2 29044.16} C_VEL
LIN {X 0,Y 607.918,Z 940.163,A -85,B 0,C 180,E1 29042.685,E2 29042.685} C_VEL
LIN {X 0,Y 607.916,Z 920.827,A -85,B 0,C 180,E1 29041.474,E2 29041.474} C_VEL
LIN {X 0,Y 607.918,Z 900.293,A -85,B 0,C 180,E1 29040.38,E2 29040.38} C_VEL
LIN {X 0,Y 607.914,Z 881.45,A -85,B 0,C 180,E1 29039.523,E2 29039.523} C_VEL
LIN {X 0,Y 607.915,Z 859.018,A -85,B 0,C 180,E1 29038.685,E2 29038.685} C_VEL
LIN {X 0,Y 607.912,Z 840.386,A -85,B 0,C 180,E1 29038.132,E2 29038.132} C_VEL
LIN {X 0,Y 607.912,Z 818.534,A -85,B 0,C 180,E1 29037.631,E2 29037.631} C_VEL
LIN {X 0,Y 607.913,Z 775.337,A -85,B 0,C 180,E1 29037.001,E2 29037.001} C_VEL
LIN {X 0,Y 607.902,Z 568.743,A -85,B 0,C 180,E1 29034.1,E2 29034.1} C_VEL
LIN {X 0,Y 607.905,Z 465.312,A -85,B 0,C 180,E1 29032.6,E2 29032.6} C_VEL
LIN {X 0,Y 607.916,Z 407.824,A -85,B 0,C 180,E1 29029.798,E2 29029.798} C_VEL
LIN {X 0,Y 607.892,Z 372.115,A -85,B 0,C 180,E1 29027.976,E2 29027.976} C_VEL
LIN {X 0,Y 607.873,Z 371.406,A -85,B 0,C 180,E1 29027.848,E2 29027.848} C_VEL
LIN {X 0,Y 607.826,Z 371.327,A -85,B 0,C 180,E1 29025.114,E2 29025.114} C_VEL
LIN {X 0,Y 607.854,Z 371.326,A -85,B 0,C 180,E1 29022.391,E2 29022.391} C_VEL
LIN {X 0,Y 607.842,Z 371.326,A -85,B 0,C 180,E1 29019.172,E2 29019.172} C_VEL
LIN {X 0,Y 607.828,Z 371.327,A -85,B 0,C 180,E1 29016.546,E2 29016.546} C_VEL
LIN {X 0,Y 607.914,Z 371.326,A -85,B 0,C 180,E1 29013.5,E2 29013.5} C_VEL
LIN {X 0,Y 607.828,Z 371.325,A -85,B 0,C 180,E1 29010.461,E2 29010.461} C_VEL
LIN {X 0,Y 607.871,Z 371.327,A -85,B 0,C 180,E1 29007.635,E2 29007.635} C_VEL
LIN {X 0,Y 607.841,Z 371.325,A -85,B 0,C 180,E1 29004.489,E2 29004.489} C_VEL
LIN {X 0,Y 607.834,Z 371.326,A -85,B 0,C 180,E1 29001.824,E2 29001.824} C_VEL
LIN {X 0,Y 607.898,Z 371.324,A -85,B 0,C 180,E1 28998.707,E2 28998.707} C_VEL
LIN {X 0,Y 607.831,Z 371.326,A -85,B 0,C 180,E1 28995.748,E2 28995.748} C_VEL
LIN {X 0,Y 607.913,Z 371.326,A -85,B 0,C 180,E1 28992.732,E2 28992.732} C_VEL
LIN {X 0,Y 607.835,Z 371.326,A -85,B 0,C 180,E1 28989.659,E2 28989.659} C_VEL
LIN {X 0,Y 607.856,Z 371.326,A -85,B 0,C 180,E1 28986.896,E2 28986.896} C_VEL
LIN {X 0,Y 607.845,Z 371.325,A -85,B 0,C 180,E1 28983.583,E2 28983.583} C_VEL
LIN {X 0,Y 607.841,Z 371.326,A -85,B 0,C 180,E1 28980.848,E2 28980.848} C_VEL
LIN {X 0,Y 607.879,Z 371.324,A -85,B 0,C 180,E1 28977.643,E2 28977.643} C_VEL
LIN {X 0,Y 607.835,Z 371.326,A -85,B 0,C 180,E1 28976.855,E2 28976.855} C_VEL
LIN {X 0,Y 606.882,Z 371.454,A -85,B 0,C 180,E1 28976.129,E2 28976.129} C_VEL
LIN {X 0,Y 600.437,Z 372.258,A -85,B 0,C 180,E1 28974.039,E2 28974.039} C_VEL
LIN {X 0,Y 599.953,Z 372.312,A -85,B 0,C 180,E1 28973.562,E2 28973.562} C_VEL
LIN {X 0,Y 599.898,Z 372.315,A -85,B 0,C 180,E1 28970.599,E2 28970.599} C_VEL
LIN {X 0,Y 599.979,Z 372.314,A -85,B 0,C 180,E1 28967.488,E2 28967.488} C_VEL
LIN {X 0,Y 599.898,Z 372.314,A -85,B 0,C 180,E1 28964.434,E2 28964.434} C_VEL
LIN {X 0,Y 599.965,Z 372.317,A -85,B 0,C 180,E1 28961.439,E2 28961.439} C_VEL
LIN {X 0,Y 599.901,Z 372.313,A -85,B 0,C 180,E1 28958.284,E2 28958.284} C_VEL
LIN {X 0,Y 599.937,Z 372.316,A -85,B 0,C 180,E1 28955.376,E2 28955.376} C_VEL
LIN {X 0,Y 599.91,Z 372.313,A -85,B 0,C 180,E1 28952.181,E2 28952.181} C_VEL
LIN {X 0,Y 599.909,Z 372.311,A -85,B 0,C 180,E1 28949.447,E2 28949.447} C_VEL
LIN {X 0,Y 599.934,Z 372.312,A -85,B 0,C 180,E1 28946.175,E2 28946.175} C_VEL
LIN {X 0,Y 599.905,Z 372.312,A -85,B 0,C 180,E1 28943.291,E2 28943.291} C_VEL
LIN {X 0,Y 599.974,Z 372.309,A -85,B 0,C 180,E1 28940.198,E2 28940.198} C_VEL
LIN {X 0,Y 599.904,Z 372.314,A -85,B 0,C 180,E1 28937.155,E2 28937.155} C_VEL
LIN {X 0,Y 599.981,Z 372.313,A -85,B 0,C 180,E1 28934.089,E2 28934.089} C_VEL
LIN {X 0,Y 599.904,Z 372.312,A -85,B 0,C 180,E1 28930.973,E2 28930.973} C_VEL
LIN {X 0,Y 599.976,Z 372.312,A -85,B 0,C 180,E1 28927.948,E2 28927.948} C_VEL
LIN {X 0,Y 599.909,Z 372.312,A -85,B 0,C 180,E1 28924.867,E2 28924.867} C_VEL
LIN {X 0,Y 599.968,Z 372.684,A -85,B 0,C 180,E1 28924.385,E2 28924.385} C_VEL
LIN {X 0,Y 600.904,Z 375.553,A -85,B 0,C 180,E1 28924.107,E2 28924.107} C_VEL
LIN {X 0,Y 600.721,Z 419.551,A -85,B 0,C 180,E1 28921.224,E2 28921.224} C_VEL
LIN {X 0,Y 600.596,Z 465.101,A -85,B 0,C 180,E1 28918.325,E2 28918.325} C_VEL
LIN {X 0,Y 600.706,Z 470.907,A -85,B 0,C 180,E1 28917.994,E2 28917.994} C_VEL
LIN {X 0,Y 600.667,Z 676.212,A -85,B 0,C 180,E1 28915.303,E2 28915.303} C_VEL
LIN {X 0,Y 600.609,Z 733.253,A -85,B 0,C 180,E1 28914.538,E2 28914.538} C_VEL
LIN {X 0,Y 600.556,Z 753.701,A -85,B 0,C 180,E1 28914.08,E2 28914.08} C_VEL
LIN {X 0,Y 600.504,Z 773.275,A -85,B 0,C 180,E1 28913.465,E2 28913.465} C_VEL
LIN {X 0,Y 600.422,Z 792.747,A -85,B 0,C 180,E1 28912.676,E2 28912.676} C_VEL
LIN {X 0,Y 600.347,Z 811.375,A -85,B 0,C 180,E1 28911.739,E2 28911.739} C_VEL
LIN {X 0,Y 600.275,Z 829.688,A -85,B 0,C 180,E1 28910.622,E2 28910.622} C_VEL
LIN {X 0,Y 600.197,Z 847.828,A -85,B 0,C 180,E1 28909.295,E2 28909.295} C_VEL
LIN {X 0,Y 600.125,Z 864.419,A -85,B 0,C 180,E1 28907.852,E2 28907.852} C_VEL
LIN {X 0,Y 600.055,Z 879.951,A -85,B 0,C 180,E1 28906.256,E2 28906.256} C_VEL
LIN {X 0,Y 600.013,Z 893.781,A -85,B 0,C 180,E1 28904.574,E2 28904.574} C_VEL
LIN {X 0,Y 599.973,Z 905.632,A -85,B 0,C 180,E1 28902.862,E2 28902.862} C_VEL
LIN {X 0,Y 599.942,Z 916.121,A -85,B 0,C 180,E1 28901.05,E2 28901.05} C_VEL
LIN {X 0,Y 599.92,Z 924.871,A -85,B 0,C 180,E1 28899.207,E2 28899.207} C_VEL
LIN {X 0,Y 599.908,Z 931.849,A -85,B 0,C 180,E1 28897.373,E2 28897.373} C_VEL
LIN {X 0,Y 599.905,Z 937.389,A -85,B 0,C 180,E1 28895.451,E2 28895.451} C_VEL
LIN {X 0,Y 599.903,Z 941.166,A -85,B 0,C 180,E1 28893.536,E2 28893.536} C_VEL
LIN {X 0,Y 599.904,Z 943.341,A -85,B 0,C 180,E1 28891.624,E2 28891.624} C_VEL
LIN {X 0,Y 599.904,Z 943.95,A -85,B 0,C 180,E1 28889.714,E2 28889.714} C_VEL
LIN {X 0,Y 599.913,Z 942.997,A -85,B 0,C 180,E1 28887.803,E2 28887.803} C_VEL
LIN {X 0,Y 599.917,Z 940.209,A -85,B 0,C 180,E1 28885.795,E2 28885.795} C_VEL
LIN {X 0,Y 599.918,Z 935.854,A -85,B 0,C 180,E1 28883.877,E2 28883.877} C_VEL
LIN {X 0,Y 599.918,Z 929.554,A -85,B 0,C 180,E1 28881.889,E2 28881.889} C_VEL
LIN {X 0,Y 599.922,Z 921.851,A -85,B 0,C 180,E1 28880.018,E2 28880.018} C_VEL
LIN {X 0,Y 599.942,Z 912.969,A -85,B 0,C 180,E1 28878.269,E2 28878.269} C_VEL
LIN {X 0,Y 599.971,Z 902.108,A -85,B 0,C 180,E1 28876.508,E2 28876.508} C_VEL
LIN {X 0,Y 600.018,Z 889.837,A -85,B 0,C 180,E1 28874.834,E2 28874.834} C_VEL
LIN {X 0,Y 600.07,Z 876.158,A -85,B 0,C 180,E1 28873.246,E2 28873.246} C_VEL
LIN {X 0,Y 600.132,Z 860.442,A -85,B 0,C 180,E1 28871.696,E2 28871.696} C_VEL
LIN {X 0,Y 600.206,Z 844.192,A -85,B 0,C 180,E1 28870.336,E2 28870.336} C_VEL
LIN {X 0,Y 600.289,Z 827.056,A -85,B 0,C 180,E1 28869.118,E2 28869.118} C_VEL
LIN {X 0,Y 600.373,Z 809.115,A -85,B 0,C 180,E1 28868.045,E2 28868.045} C_VEL
LIN {X 0,Y 600.434,Z 790.217,A -85,B 0,C 180,E1 28867.118,E2 28867.118} C_VEL
LIN {X 0,Y 600.506,Z 771.103,A -85,B 0,C 180,E1 28866.368,E2 28866.368} C_VEL
LIN {X 0,Y 600.563,Z 750.423,A -85,B 0,C 180,E1 28865.748,E2 28865.748} C_VEL
LIN {X 0,Y 600.615,Z 730.361,A -85,B 0,C 180,E1 28865.325,E2 28865.325} C_VEL
LIN {X 0,Y 600.769,Z 471.35,A -85,B 0,C 180,E1 28861.926,E2 28861.926} C_VEL
LIN {X 0,Y 600.576,Z 468.256,A -85,B 0,C 180,E1 28861.783,E2 28861.783} C_VEL
LIN {X 0,Y 600.707,Z 423.441,A -85,B 0,C 180,E1 28858.936,E2 28858.936} C_VEL
LIN {X 0,Y 600.903,Z 378.624,A -85,B 0,C 180,E1 28856.008,E2 28856.008} C_VEL
LIN {X 0,Y 600.859,Z 375.176,A -85,B 0,C 180,E1 28855.774,E2 28855.774} C_VEL
LIN {X 0,Y 599.944,Z 372.512,A -85,B 0,C 180,E1 28855.483,E2 28855.483} C_VEL
LIN {X 0,Y 599.938,Z 372.311,A -85,B 0,C 180,E1 28852.652,E2 28852.652} C_VEL
LIN {X 0,Y 599.929,Z 372.313,A -85,B 0,C 180,E1 28849.459,E2 28849.459} C_VEL
LIN {X 0,Y 599.927,Z 372.312,A -85,B 0,C 180,E1 28846.502,E2 28846.502} C_VEL
LIN {X 0,Y 599.932,Z 372.315,A -85,B 0,C 180,E1 28843.234,E2 28843.234} C_VEL
LIN {X 0,Y 599.921,Z 372.31,A -85,B 0,C 180,E1 28840.291,E2 28840.291} C_VEL
LIN {X 0,Y 599.933,Z 372.313,A -85,B 0,C 180,E1 28836.988,E2 28836.988} C_VEL
LIN {X 0,Y 599.917,Z 372.312,A -85,B 0,C 180,E1 28834.056,E2 28834.056} C_VEL
LIN {X 0,Y 599.937,Z 372.312,A -85,B 0,C 180,E1 28830.774,E2 28830.774} C_VEL
LIN {X 0,Y 599.908,Z 372.313,A -85,B 0,C 180,E1 28827.927,E2 28827.927} C_VEL
LIN {X 0,Y 599.971,Z 372.316,A -85,B 0,C 180,E1 28824.832,E2 28824.832} C_VEL
LIN {X 0,Y 599.905,Z 372.313,A -85,B 0,C 180,E1 28821.819,E2 28821.819} C_VEL
LIN {X 0,Y 599.976,Z 372.313,A -85,B 0,C 180,E1 28818.762,E2 28818.762} C_VEL
LIN {X 0,Y 599.904,Z 372.314,A -85,B 0,C 180,E1 28815.665,E2 28815.665} C_VEL
LIN {X 0,Y 599.957,Z 372.312,A -85,B 0,C 180,E1 28812.708,E2 28812.708} C_VEL
LIN {X 0,Y 599.909,Z 372.315,A -85,B 0,C 180,E1 28809.594,E2 28809.594} C_VEL
LIN {X 0,Y 599.916,Z 372.312,A -85,B 0,C 180,E1 28806.796,E2 28806.796} C_VEL
LIN {X 0,Y 599.915,Z 372.315,A -85,B 0,C 180,E1 28803.44,E2 28803.44} C_VEL
LIN {X 0,Y 599.906,Z 372.314,A -85,B 0,C 180,E1 28800.669,E2 28800.669} C_VEL
LIN {X 0,Y 599.938,Z 372.316,A -85,B 0,C 180,E1 28797.421,E2 28797.421} C_VEL
LIN {X 0,Y 599.899,Z 372.314,A -85,B 0,C 180,E1 28794.549,E2 28794.549} C_VEL
LIN {X 0,Y 599.978,Z 372.315,A -85,B 0,C 180,E1 28791.471,E2 28791.471} C_VEL
LIN {X 0,Y 599.896,Z 372.313,A -85,B 0,C 180,E1 28788.463,E2 28788.463} C_VEL
LIN {X 0,Y 599.951,Z 372.31,A -85,B 0,C 180,E1 28785.531,E2 28785.531} C_VEL
LIN {X 0,Y 599.898,Z 372.314,A -85,B 0,C 180,E1 28782.342,E2 28782.342} C_VEL
LIN {X 0,Y 599.919,Z 372.311,A -85,B 0,C 180,E1 28779.513,E2 28779.513} C_VEL
LIN {X 0,Y 599.904,Z 372.315,A -85,B 0,C 180,E1 28776.209,E2 28776.209} C_VEL
LIN {X 0,Y 599.9,Z 372.313,A -85,B 0,C 180,E1 28773.47,E2 28773.47} C_VEL
LIN {X 0,Y 599.928,Z 372.313,A -85,B 0,C 180,E1 28770.221,E2 28770.221} C_VEL
LIN {X 0,Y 599.891,Z 372.316,A -85,B 0,C 180,E1 28767.429,E2 28767.429} C_VEL
LIN {X 0,Y 599.973,Z 372.313,A -85,B 0,C 180,E1 28764.416,E2 28764.416} C_VEL
LIN {X 0,Y 599.892,Z 372.314,A -85,B 0,C 180,E1 28761.417,E2 28761.417} C_VEL
LIN {X 0,Y 599.906,Z 372.317,A -85,B 0,C 180,E1 28758.7,E2 28758.7} C_VEL
LIN {X 0,Y 599.903,Z 372.318,A -85,B 0,C 180,E1 28755.372,E2 28755.372} C_VEL
LIN {X 0,Y 599.903,Z 372.423,A -85,B 0,C 180,E1 28752.778,E2 28752.778} C_VEL
LIN {X 0,Y 600.227,Z 373.798,A -85,B 0,C 180,E1 28752.585,E2 28752.585} C_VEL
LIN {X 0,Y 601.639,Z 376.794,A -85,B 0,C 180,E1 28752.305,E2 28752.305} C_VEL
LIN {X 0,Y 601.435,Z 433.668,A -85,B 0,C 180,E1 28749.425,E2 28749.425} C_VEL
LIN {X 0,Y 601.458,Z 466.253,A -85,B 0,C 180,E1 28747.849,E2 28747.849} C_VEL
LIN {X 0,Y 601.325,Z 654.497,A -85,B 0,C 180,E1 28745.118,E2 28745.118} C_VEL
LIN {X 0,Y 601.147,Z 815.219,A -85,B 0,C 180,E1 28742.833,E2 28742.833} C_VEL
LIN {X 0,Y 601.067,Z 838.899,A -85,B 0,C 180,E1 28742.315,E2 28742.315} C_VEL
LIN {X 0,Y 601.002,Z 858.222,A -85,B 0,C 180,E1 28741.743,E2 28741.743} C_VEL
LIN {X 0,Y 600.878,Z 880.547,A -85,B 0,C 180,E1 28740.912,E2 28740.912} C_VEL
LIN {X 0,Y 600.793,Z 900.297,A -85,B 0,C 180,E1 28740.007,E2 28740.007} C_VEL
LIN {X 0,Y 600.656,Z 921.465,A -85,B 0,C 180,E1 28738.865,E2 28738.865} C_VEL
LIN {X 0,Y 600.559,Z 940.89,A -85,B 0,C 180,E1 28737.63,E2 28737.63} C_VEL
LIN {X 0,Y 600.418,Z 960.952,A -85,B 0,C 180,E1 28736.159,E2 28736.159} C_VEL
LIN {X 0,Y 600.324,Z 979.725,A -85,B 0,C 180,E1 28734.581,E2 28734.581} C_VEL
LIN {X 0,Y 600.218,Z 997.052,A -85,B 0,C 180,E1 28732.899,E2 28732.899} C_VEL
LIN {X 0,Y 600.135,Z 1014.283,A -85,B 0,C 180,E1 28730.99,E2 28730.99} C_VEL
LIN {X 0,Y 600.074,Z 1028.96,A -85,B 0,C 180,E1 28729.136,E2 28729.136} C_VEL
LIN {X 0,Y 600.014,Z 1042.446,A -85,B 0,C 180,E1 28727.155,E2 28727.155} C_VEL
LIN {X 0,Y 599.975,Z 1054.748,A -85,B 0,C 180,E1 28725.069,E2 28725.069} C_VEL
LIN {X 0,Y 599.925,Z 1064.147,A -85,B 0,C 180,E1 28723.199,E2 28723.199} C_VEL
LIN {X 0,Y 599.91,Z 1073.267,A -85,B 0,C 180,E1 28721.05,E2 28721.05} C_VEL
LIN {X 0,Y 599.92,Z 1079.952,A -85,B 0,C 180,E1 28719.11,E2 28719.11} C_VEL
LIN {X 0,Y 599.885,Z 1085.807,A -85,B 0,C 180,E1 28716.989,E2 28716.989} C_VEL
LIN {X 0,Y 599.907,Z 1089.798,A -85,B 0,C 180,E1 28714.972,E2 28714.972} C_VEL
LIN {X 0,Y 599.892,Z 1092.63,A -85,B 0,C 180,E1 28712.866,E2 28712.866} C_VEL
LIN {X 0,Y 599.883,Z 1093.828,A -85,B 0,C 180,E1 28710.764,E2 28710.764} C_VEL
LIN {X 0,Y 599.914,Z 1093.694,A -85,B 0,C 180,E1 28708.663,E2 28708.663} C_VEL
LIN {X 0,Y 599.886,Z 1091.953,A -85,B 0,C 180,E1 28706.56,E2 28706.56} C_VEL
LIN {X 0,Y 599.899,Z 1089.001,A -85,B 0,C 180,E1 28704.548,E2 28704.548} C_VEL
LIN {X 0,Y 599.914,Z 1084.08,A -85,B 0,C 180,E1 28702.338,E2 28702.338} C_VEL
LIN {X 0,Y 599.893,Z 1078.428,A -85,B 0,C 180,E1 28700.405,E2 28700.405} C_VEL
LIN {X 0,Y 599.925,Z 1070.148,A -85,B 0,C 180,E1 28698.171,E2 28698.171} C_VEL
LIN {X 0,Y 599.934,Z 1061.827,A -85,B 0,C 180,E1 28696.31,E2 28696.31} C_VEL
LIN {X 0,Y 599.967,Z 1050.294,A -85,B 0,C 180,E1 28694.139,E2 28694.139} C_VEL
LIN {X 0,Y 600.009,Z 1038.588,A -85,B 0,C 180,E1 28692.245,E2 28692.245} C_VEL
LIN {X 0,Y 600.079,Z 1024.551,A -85,B 0,C 180,E1 28690.288,E2 28690.288} C_VEL
LIN {X 0,Y 600.164,Z 1009.517,A -85,B 0,C 180,E1 28688.448,E2 28688.448} C_VEL
LIN {X 0,Y 600.237,Z 993.073,A -85,B 0,C 180,E1 28686.695,E2 28686.695} C_VEL
LIN {X 0,Y 600.348,Z 975.207,A -85,B 0,C 180,E1 28685.026,E2 28685.026} C_VEL
LIN {X 0,Y 600.471,Z 956.596,A -85,B 0,C 180,E1 28683.496,E2 28683.496} C_VEL
LIN {X 0,Y 600.565,Z 936.956,A -85,B 0,C 180,E1 28682.106,E2 28682.106} C_VEL
LIN {X 0,Y 600.707,Z 915.787,A -85,B 0,C 180,E1 28680.811,E2 28680.811} C_VEL
LIN {X 0,Y 600.801,Z 895.711,A -85,B 0,C 180,E1 28679.767,E2 28679.767} C_VEL
LIN {X 0,Y 600.936,Z 872.851,A -85,B 0,C 180,E1 28678.782,E2 28678.782} C_VEL
LIN {X 0,Y 601.01,Z 853.099,A -85,B 0,C 180,E1 28678.091,E2 28678.091} C_VEL
LIN {X 0,Y 601.109,Z 829.394,A -85,B 0,C 180,E1 28677.453,E2 28677.453} C_VEL
LIN {X 0,Y 601.154,Z 810.187,A -85,B 0,C 180,E1 28677.084,E2 28677.084} C_VEL
LIN {X 0,Y 601.413,Z 584.406,A -85,B 0,C 180,E1 28673.879,E2 28673.879} C_VEL
LIN {X 0,Y 601.386,Z 465.601,A -85,B 0,C 180,E1 28672.131,E2 28672.131} C_VEL
LIN {X 0,Y 601.536,Z 406.466,A -85,B 0,C 180,E1 28669.214,E2 28669.214} C_VEL
LIN {X 0,Y 601.574,Z 376.283,A -85,B 0,C 180,E1 28667.663,E2 28667.663} C_VEL
LIN {X 0,Y 599.958,Z 372.757,A -85,B 0,C 180,E1 28667.302,E2 28667.302} C_VEL
LIN {X 0,Y 599.887,Z 372.296,A -85,B 0,C 180,E1 28667.023,E2 28667.023} C_VEL
LIN {X 0,Y 599.976,Z 372.312,A -85,B 0,C 180,E1 28663.951,E2 28663.951} C_VEL
LIN {X 0,Y 599.889,Z 372.317,A -85,B 0,C 180,E1 28660.921,E2 28660.921} C_VEL
LIN {X 0,Y 599.925,Z 372.315,A -85,B 0,C 180,E1 28658.125,E2 28658.125} C_VEL
LIN {X 0,Y 599.899,Z 372.314,A -85,B 0,C 180,E1 28654.912,E2 28654.912} C_VEL
LIN {X 0,Y 599.896,Z 372.316,A -85,B 0,C 180,E1 28652.232,E2 28652.232} C_VEL
LIN {X 0,Y 599.935,Z 372.315,A -85,B 0,C 180,E1 28649.011,E2 28649.011} C_VEL
LIN {X 0,Y 599.891,Z 372.314,A -85,B 0,C 180,E1 28646.105,E2 28646.105} C_VEL
LIN {X 0,Y 599.974,Z 372.316,A -85,B 0,C 180,E1 28643.055,E2 28643.055} C_VEL
LIN {X 0,Y 599.893,Z 372.312,A -85,B 0,C 180,E1 28640.08,E2 28640.08} C_VEL
LIN {X 0,Y 599.926,Z 372.315,A -85,B 0,C 180,E1 28637.255,E2 28637.255} C_VEL
LIN {X 0,Y 599.907,Z 372.312,A -85,B 0,C 180,E1 28634.065,E2 28634.065} C_VEL
LIN {X 0,Y 599.898,Z 372.314,A -85,B 0,C 180,E1 28631.342,E2 28631.342} C_VEL
LIN {X 0,Y 599.944,Z 372.313,A -85,B 0,C 180,E1 28628.144,E2 28628.144} C_VEL
LIN {X 0,Y 599.894,Z 372.315,A -85,B 0,C 180,E1 28625.259,E2 28625.259} C_VEL
LIN {X 0,Y 599.976,Z 372.315,A -85,B 0,C 180,E1 28622.196,E2 28622.196} C_VEL
LIN {X 0,Y 599.897,Z 372.314,A -85,B 0,C 180,E1 28619.14,E2 28619.14} C_VEL
LIN {X 0,Y 599.937,Z 372.316,A -85,B 0,C 180,E1 28616.273,E2 28616.273} C_VEL
LIN {X 0,Y 599.953,Z 372.312,A -85,B 0,C 180,E1 28613.562,E2 28613.562} C_VEL
LIN {X 0,Y 598.887,Z 372.443,A -85,B 0,C 180,E1 28612.826,E2 28612.826} C_VEL
LIN {X 0,Y 592.469,Z 373.242,A -85,B 0,C 180,E1 28610.762,E2 28610.762} C_VEL
LIN {X 0,Y 591.977,Z 373.305,A -85,B 0,C 180,E1 28610.225,E2 28610.225} C_VEL
LIN {X 0,Y 591.976,Z 373.303,A -85,B 0,C 180,E1 28606.919,E2 28606.919} C_VEL
LIN {X 0,Y 591.967,Z 373.303,A -85,B 0,C 180,E1 28604.12,E2 28604.12} C_VEL
LIN {X 0,Y 591.999,Z 373.302,A -85,B 0,C 180,E1 28600.873,E2 28600.873} C_VEL
LIN {X 0,Y 591.963,Z 373.303,A -85,B 0,C 180,E1 28597.977,E2 28597.977} C_VEL
LIN {X 0,Y 592.028,Z 373.301,A -85,B 0,C 180,E1 28594.811,E2 28594.811} C_VEL
LIN {X 0,Y 591.963,Z 373.303,A -85,B 0,C 180,E1 28591.775,E2 28591.775} C_VEL
LIN {X 0,Y 592.037,Z 373.302,A -85,B 0,C 180,E1 28588.656,E2 28588.656} C_VEL
LIN {X 0,Y 591.963,Z 373.303,A -85,B 0,C 180,E1 28585.54,E2 28585.54} C_VEL
LIN {X 0,Y 592.04,Z 373.302,A -85,B 0,C 180,E1 28582.379,E2 28582.379} C_VEL
LIN {X 0,Y 591.965,Z 373.3,A -85,B 0,C 180,E1 28579.309,E2 28579.309} C_VEL
LIN {X 0,Y 592.042,Z 373.3,A -85,B 0,C 180,E1 28576.148,E2 28576.148} C_VEL
LIN {X 0,Y 591.966,Z 373.304,A -85,B 0,C 180,E1 28573.03,E2 28573.03} C_VEL
LIN {X 0,Y 592.038,Z 373.301,A -85,B 0,C 180,E1 28569.924,E2 28569.924} C_VEL
LIN {X 0,Y 591.966,Z 373.303,A -85,B 0,C 180,E1 28566.811,E2 28566.811} C_VEL
LIN {X 0,Y 591.983,Z 373.383,A -85,B 0,C 180,E1 28564.93,E2 28564.93} C_VEL
LIN {X 0,Y 592.089,Z 374.009,A -85,B 0,C 180,E1 28564.805,E2 28564.805} C_VEL
LIN {X 0,Y 593.915,Z 379.008,A -85,B 0,C 180,E1 28564.331,E2 28564.331} C_VEL
LIN {X 0,Y 593.566,Z 422.92,A -85,B 0,C 180,E1 28561.423,E2 28561.423} C_VEL
LIN {X 0,Y 593.302,Z 467.696,A -85,B 0,C 180,E1 28558.54,E2 28558.54} C_VEL
LIN {X 0,Y 593.442,Z 471.071,A -85,B 0,C 180,E1 28558.365,E2 28558.365} C_VEL
LIN {X 0,Y 593.729,Z 477.781,A -85,B 0,C 180,E1 28558.26,E2 28558.26} C_VEL
LIN {X 0,Y 593.333,Z 732.571,A -85,B 0,C 180,E1 28554.873,E2 28554.873} C_VEL
LIN {X 0,Y 593.228,Z 752.871,A -85,B 0,C 180,E1 28554.419,E2 28554.419} C_VEL
LIN {X 0,Y 593.111,Z 772.252,A -85,B 0,C 180,E1 28553.813,E2 28553.813} C_VEL
LIN {X 0,Y 592.955,Z 791.646,A -85,B 0,C 180,E1 28553.03,E2 28553.03} C_VEL
LIN {X 0,Y 592.82,Z 810.272,A -85,B 0,C 180,E1 28552.093,E2 28552.093} C_VEL
LIN {X 0,Y 592.662,Z 828.862,A -85,B 0,C 180,E1 28550.957,E2 28550.957} C_VEL
LIN {X 0,Y 592.498,Z 846.378,A -85,B 0,C 180,E1 28549.67,E2 28549.67} C_VEL
LIN {X 0,Y 592.349,Z 862.22,A -85,B 0,C 180,E1 28548.298,E2 28548.298} C_VEL
LIN {X 0,Y 592.225,Z 877.181,A -85,B 0,C 180,E1 28546.78,E2 28546.78} C_VEL
LIN {X 0,Y 592.125,Z 890.689,A -85,B 0,C 180,E1 28545.173,E2 28545.173} C_VEL
LIN {X 0,Y 592.032,Z 903.322,A -85,B 0,C 180,E1 28543.397,E2 28543.397} C_VEL
LIN {X 0,Y 591.979,Z 913.535,A -85,B 0,C 180,E1 28541.694,E2 28541.694} C_VEL
LIN {X 0,Y 591.943,Z 922.807,A -85,B 0,C 180,E1 28539.823,E2 28539.823} C_VEL
LIN {X 0,Y 591.924,Z 930.164,A -85,B 0,C 180,E1 28537.962,E2 28537.962} C_VEL
LIN {X 0,Y 591.918,Z 936.125,A -85,B 0,C 180,E1 28536.012,E2 28536.012} C_VEL
LIN {X 0,Y 591.916,Z 940.378,A -85,B 0,C 180,E1 28534.068,E2 28534.068} C_VEL
LIN {X 0,Y 591.915,Z 943.002,A -85,B 0,C 180,E1 28532.13,E2 28532.13} C_VEL
LIN {X 0,Y 591.912,Z 943.974,A -85,B 0,C 180,E1 28530.097,E2 28530.097} C_VEL
LIN {X 0,Y 591.911,Z 943.271,A -85,B 0,C 180,E1 28528.161,E2 28528.161} C_VEL
LIN {X 0,Y 591.915,Z 940.84,A -85,B 0,C 180,E1 28526.126,E2 28526.126} C_VEL
LIN {X 0,Y 591.921,Z 936.612,A -85,B 0,C 180,E1 28524.086,E2 28524.086} C_VEL
LIN {X 0,Y 591.932,Z 931.197,A -85,B 0,C 180,E1 28522.234,E2 28522.234} C_VEL
LIN {X 0,Y 591.943,Z 923.621,A -85,B 0,C 180,E1 28520.275,E2 28520.275} C_VEL
LIN {X 0,Y 591.973,Z 914.525,A -85,B 0,C 180,E1 28518.405,E2 28518.405} C_VEL
LIN {X 0,Y 592.03,Z 903.906,A -85,B 0,C 180,E1 28516.603,E2 28516.603} C_VEL
LIN {X 0,Y 592.119,Z 891.385,A -85,B 0,C 180,E1 28514.827,E2 28514.827} C_VEL
LIN {X 0,Y 592.224,Z 877.745,A -85,B 0,C 180,E1 28513.191,E2 28513.191} C_VEL
LIN {X 0,Y 592.344,Z 863.197,A -85,B 0,C 180,E1 28511.702,E2 28511.702} C_VEL
LIN {X 0,Y 592.498,Z 846.83,A -85,B 0,C 180,E1 28510.275,E2 28510.275} C_VEL
LIN {X 0,Y 592.657,Z 829.428,A -85,B 0,C 180,E1 28508.991,E2 28508.991} C_VEL
LIN {X 0,Y 592.808,Z 810.923,A -85,B 0,C 180,E1 28507.854,E2 28507.854} C_VEL
LIN {X 0,Y 592.951,Z 792.45,A -85,B 0,C 180,E1 28506.918,E2 28506.918} C_VEL
LIN {X 0,Y 593.109,Z 772.557,A -85,B 0,C 180,E1 28506.108,E2 28506.108} C_VEL
LIN {X 0,Y 593.23,Z 752.478,A -85,B 0,C 180,E1 28505.481,E2 28505.481} C_VEL
LIN {X 0,Y 593.334,Z 732.356,A -85,B 0,C 180,E1 28505.033,E2 28505.033} C_VEL
LIN {X 0,Y 593.723,Z 477.413,A -85,B 0,C 180,E1 28501.645,E2 28501.645} C_VEL
LIN {X 0,Y 593.446,Z 471.125,A -85,B 0,C 180,E1 28501.546,E2 28501.546} C_VEL
LIN {X 0,Y 593.302,Z 467.383,A -85,B 0,C 180,E1 28501.35,E2 28501.35} C_VEL
LIN {X 0,Y 593.607,Z 419.983,A -85,B 0,C 180,E1 28498.296,E2 28498.296} C_VEL
LIN {X 0,Y 593.864,Z 378.612,A -85,B 0,C 180,E1 28495.548,E2 28495.548} C_VEL
LIN {X 0,Y 592.047,Z 373.744,A -85,B 0,C 180,E1 28495.074,E2 28495.074} C_VEL
LIN {X 0,Y 592.003,Z 373.299,A -85,B 0,C 180,E1 28494.716,E2 28494.716} C_VEL
LIN {X 0,Y 591.984,Z 373.306,A -85,B 0,C 180,E1 28491.445,E2 28491.445} C_VEL
LIN {X 0,Y 591.992,Z 373.298,A -85,B 0,C 180,E1 28488.541,E2 28488.541} C_VEL
LIN {X 0,Y 591.983,Z 373.302,A -85,B 0,C 180,E1 28485.185,E2 28485.185} C_VEL
LIN {X 0,Y 591.994,Z 373.301,A -85,B 0,C 180,E1 28482.238,E2 28482.238} C_VEL
LIN {X 0,Y 591.983,Z 373.304,A -85,B 0,C 180,E1 28478.926,E2 28478.926} C_VEL
LIN {X 0,Y 591.989,Z 373.297,A -85,B 0,C 180,E1 28475.999,E2 28475.999} C_VEL
LIN {X 0,Y 591.986,Z 373.304,A -85,B 0,C 180,E1 28472.716,E2 28472.716} C_VEL
LIN {X 0,Y 591.976,Z 373.296,A -85,B 0,C 180,E1 28469.885,E2 28469.885} C_VEL
LIN {X 0,Y 591.996,Z 373.304,A -85,B 0,C 180,E1 28466.588,E2 28466.588} C_VEL
LIN {X 0,Y 591.972,Z 373.302,A -85,B 0,C 180,E1 28463.703,E2 28463.703} C_VEL
LIN {X 0,Y 592.011,Z 373.305,A -85,B 0,C 180,E1 28460.464,E2 28460.464} C_VEL
LIN {X 0,Y 591.967,Z 373.302,A -85,B 0,C 180,E1 28457.497,E2 28457.497} C_VEL
LIN {X 0,Y 592.033,Z 373.305,A -85,B 0,C 180,E1 28454.375,E2 28454.375} C_VEL
LIN {X 0,Y 591.963,Z 373.302,A -85,B 0,C 180,E1 28451.398,E2 28451.398} C_VEL
LIN {X 0,Y 592.038,Z 373.302,A -85,B 0,C 180,E1 28448.351,E2 28448.351} C_VEL
LIN {X 0,Y 591.963,Z 373.304,A -85,B 0,C 180,E1 28445.233,E2 28445.233} C_VEL
LIN {X 0,Y 592.019,Z 373.301,A -85,B 0,C 180,E1 28442.226,E2 28442.226} C_VEL
LIN {X 0,Y 591.963,Z 373.304,A -85,B 0,C 180,E1 28439.033,E2 28439.033} C_VEL
LIN {X 0,Y 591.996,Z 373.302,A -85,B 0,C 180,E1 28436.127,E2 28436.127} C_VEL
LIN {X 0,Y 591.969,Z 373.303,A -85,B 0,C 180,E1 28432.918,E2 28432.918} C_VEL
LIN {X 0,Y 591.974,Z 373.303,A -85,B 0,C 180,E1 28430.08,E2 28430.08} C_VEL
LIN {X 0,Y 591.972,Z 373.3,A -85,B 0,C 180,E1 28426.72,E2 28426.72} C_VEL
LIN {X 0,Y 591.965,Z 373.303,A -85,B 0,C 180,E1 28423.919,E2 28423.919} C_VEL
LIN {X 0,Y 591.99,Z 373.3,A -85,B 0,C 180,E1 28420.668,E2 28420.668} C_VEL
LIN {X 0,Y 591.955,Z 373.304,A -85,B 0,C 180,E1 28417.873,E2 28417.873} C_VEL
LIN {X 0,Y 592.034,Z 373.3,A -85,B 0,C 180,E1 28414.812,E2 28414.812} C_VEL
LIN {X 0,Y 591.954,Z 373.305,A -85,B 0,C 180,E1 28411.775,E2 28411.775} C_VEL
LIN {X 0,Y 591.997,Z 373.299,A -85,B 0,C 180,E1 28408.881,E2 28408.881} C_VEL
LIN {X 0,Y 591.957,Z 373.303,A -85,B 0,C 180,E1 28405.657,E2 28405.657} C_VEL
LIN {X 0,Y 591.966,Z 373.305,A -85,B 0,C 180,E1 28402.916,E2 28402.916} C_VEL
LIN {X 0,Y 591.966,Z 373.307,A -85,B 0,C 180,E1 28399.565,E2 28399.565} C_VEL
LIN {X 0,Y 591.952,Z 373.299,A -85,B 0,C 180,E1 28396.837,E2 28396.837} C_VEL
LIN {X 0,Y 592.006,Z 373.274,A -85,B 0,C 180,E1 28393.692,E2 28393.692} C_VEL
LIN {X 0,Y 592.034,Z 373.715,A -85,B 0,C 180,E1 28393.361,E2 28393.361} C_VEL
LIN {X 0,Y 593.459,Z 377.058,A -85,B 0,C 180,E1 28393.013,E2 28393.013} C_VEL
LIN {X 0,Y 594.681,Z 379.266,A -85,B 0,C 180,E1 28392.786,E2 28392.786} C_VEL
LIN {X 0,Y 595.394,Z 380.69,A -85,B 0,C 180,E1 28392.647,E2 28392.647} C_VEL
LIN {X 0,Y 594.966,Z 437.377,A -85,B 0,C 180,E1 28389.751,E2 28389.751} C_VEL
LIN {X 0,Y 594.922,Z 466.341,A -85,B 0,C 180,E1 28388.338,E2 28388.338} C_VEL
LIN {X 0,Y 595.198,Z 472.553,A -85,B 0,C 180,E1 28388.223,E2 28388.223} C_VEL
LIN {X 0,Y 594.735,Z 677.534,A -85,B 0,C 180,E1 28385.232,E2 28385.232} C_VEL
LIN {X 0,Y 594.412,Z 815.433,A -85,B 0,C 180,E1 28383.25,E2 28383.25} C_VEL
LIN {X 0,Y 594.25,Z 839.133,A -85,B 0,C 180,E1 28382.725,E2 28382.725} C_VEL
LIN {X 0,Y 594.114,Z 859.025,A -85,B 0,C 180,E1 28382.128,E2 28382.128} C_VEL
LIN {X 0,Y 593.861,Z 882.395,A -85,B 0,C 180,E1 28381.236,E2 28381.236} C_VEL
LIN {X 0,Y 593.682,Z 902.537,A -85,B 0,C 180,E1 28380.292,E2 28380.292} C_VEL
LIN {X 0,Y 593.399,Z 924.139,A -85,B 0,C 180,E1 28379.086,E2 28379.086} C_VEL
LIN {X 0,Y 593.199,Z 944.434,A -85,B 0,C 180,E1 28377.761,E2 28377.761} C_VEL
LIN {X 0,Y 592.93,Z 963.255,A -85,B 0,C 180,E1 28376.327,E2 28376.327} C_VEL
LIN {X 0,Y 592.699,Z 982.325,A -85,B 0,C 180,E1 28374.671,E2 28374.671} C_VEL
LIN {X 0,Y 592.528,Z 999.335,A -85,B 0,C 180,E1 28372.976,E2 28372.976} C_VEL
LIN {X 0,Y 592.358,Z 1015.136,A -85,B 0,C 180,E1 28371.175,E2 28371.175} C_VEL
LIN {X 0,Y 592.233,Z 1029.59,A -85,B 0,C 180,E1 28369.31,E2 28369.31} C_VEL
LIN {X 0,Y 592.123,Z 1042.448,A -85,B 0,C 180,E1 28367.391,E2 28367.391} C_VEL
LIN {X 0,Y 592.031,Z 1054.75,A -85,B 0,C 180,E1 28365.276,E2 28365.276} C_VEL
LIN {X 0,Y 591.962,Z 1064.186,A -85,B 0,C 180,E1 28363.372,E2 28363.372} C_VEL
LIN {X 0,Y 591.931,Z 1073.268,A -85,B 0,C 180,E1 28361.201,E2 28361.201} C_VEL
LIN {X 0,Y 591.918,Z 1079.953,A -85,B 0,C 180,E1 28359.234,E2 28359.234} C_VEL
LIN {X 0,Y 591.888,Z 1085.807,A -85,B 0,C 180,E1 28357.084,E2 28357.084} C_VEL
LIN {X 0,Y 591.91,Z 1089.798,A -85,B 0,C 180,E1 28355.039,E2 28355.039} C_VEL
LIN {X 0,Y 591.89,Z 1092.63,A -85,B 0,C 180,E1 28352.905,E2 28352.905} C_VEL
LIN {X 0,Y 591.884,Z 1093.828,A -85,B 0,C 180,E1 28350.774,E2 28350.774} C_VEL
LIN {X 0,Y 591.914,Z 1093.694,A -85,B 0,C 180,E1 28348.645,E2 28348.645} C_VEL
LIN {X 0,Y 591.888,Z 1091.953,A -85,B 0,C 180,E1 28346.513,E2 28346.513} C_VEL
LIN {X 0,Y 591.896,Z 1089.002,A -85,B 0,C 180,E1 28344.475,E2 28344.475} C_VEL
LIN {X 0,Y 591.925,Z 1084.08,A -85,B 0,C 180,E1 28342.234,E2 28342.234} C_VEL
LIN {X 0,Y 591.903,Z 1078.428,A -85,B 0,C 180,E1 28340.275,E2 28340.275} C_VEL
LIN {X 0,Y 591.947,Z 1070.149,A -85,B 0,C 180,E1 28338.009,E2 28338.009} C_VEL
LIN {X 0,Y 591.986,Z 1061.829,A -85,B 0,C 180,E1 28336.123,E2 28336.123} C_VEL
LIN {X 0,Y 592.052,Z 1050.296,A -85,B 0,C 180,E1 28333.921,E2 28333.921} C_VEL
LIN {X 0,Y 592.134,Z 1038.59,A -85,B 0,C 180,E1 28332,E2 28332} C_VEL
LIN {X 0,Y 592.253,Z 1024.883,A -85,B 0,C 180,E1 28330.061,E2 28330.061} C_VEL
LIN {X 0,Y 592.42,Z 1009.633,A -85,B 0,C 180,E1 28328.165,E2 28328.165} C_VEL
LIN {X 0,Y 592.569,Z 993.579,A -85,B 0,C 180,E1 28326.428,E2 28326.428} C_VEL
LIN {X 0,Y 592.797,Z 975.32,A -85,B 0,C 180,E1 28324.696,E2 28324.696} C_VEL
LIN {X 0,Y 593.043,Z 956.596,A -85,B 0,C 180,E1 28323.138,E2 28323.138} C_VEL
LIN {X 0,Y 593.242,Z 936.959,A -85,B 0,C 180,E1 28321.731,E2 28321.731} C_VEL
LIN {X 0,Y 593.532,Z 914.848,A -85,B 0,C 180,E1 28320.371,E2 28320.371} C_VEL
LIN {X 0,Y 593.732,Z 894.708,A -85,B 0,C 180,E1 28319.319,E2 28319.319} C_VEL
LIN {X 0,Y 593.987,Z 872.196,A -85,B 0,C 180,E1 28318.35,E2 28318.35} C_VEL
LIN {X 0,Y 594.145,Z 851.265,A -85,B 0,C 180,E1 28317.617,E2 28317.617} C_VEL
LIN {X 0,Y 594.335,Z 828.391,A -85,B 0,C 180,E1 28317.013,E2 28317.013} C_VEL
LIN {X 0,Y 594.431,Z 808.69,A -85,B 0,C 180,E1 28316.638,E2 28316.638} C_VEL
LIN {X 0,Y 594.94,Z 587.054,A -85,B 0,C 180,E1 28313.462,E2 28313.462} C_VEL
LIN {X 0,Y 595.027,Z 467.054,A -85,B 0,C 180,E1 28311.681,E2 28311.681} C_VEL
LIN {X 0,Y 594.8,Z 462.104,A -85,B 0,C 180,E1 28311.478,E2 28311.478} C_VEL
LIN {X 0,Y 595.227,Z 403.226,A -85,B 0,C 180,E1 28308.519,E2 28308.519} C_VEL
LIN {X 0,Y 595.395,Z 380.685,A -85,B 0,C 180,E1 28307.352,E2 28307.352} C_VEL
LIN {X 0,Y 594.004,Z 377.736,A -85,B 0,C 180,E1 28307.072,E2 28307.072} C_VEL
LIN {X 0,Y 592.151,Z 374.284,A -85,B 0,C 180,E1 28306.715,E2 28306.715} C_VEL
LIN {X 0,Y 591.987,Z 373.33,A -85,B 0,C 180,E1 28306.513,E2 28306.513} C_VEL
LIN {X 0,Y 591.958,Z 373.299,A -85,B 0,C 180,E1 28303.281,E2 28303.281} C_VEL
LIN {X 0,Y 591.959,Z 373.307,A -85,B 0,C 180,E1 28300.528,E2 28300.528} C_VEL
LIN {X 0,Y 591.984,Z 373.305,A -85,B 0,C 180,E1 28297.295,E2 28297.295} C_VEL
LIN {X 0,Y 591.952,Z 373.303,A -85,B 0,C 180,E1 28294.46,E2 28294.46} C_VEL
LIN {X 0,Y 592.028,Z 373.299,A -85,B 0,C 180,E1 28291.343,E2 28291.343} C_VEL
LIN {X 0,Y 591.952,Z 373.305,A -85,B 0,C 180,E1 28288.335,E2 28288.335} C_VEL
LIN {X 0,Y 592.023,Z 373.3,A -85,B 0,C 180,E1 28285.295,E2 28285.295} C_VEL
LIN {X 0,Y 591.956,Z 373.304,A -85,B 0,C 180,E1 28282.231,E2 28282.231} C_VEL
LIN {X 0,Y 591.976,Z 373.3,A -85,B 0,C 180,E1 28279.435,E2 28279.435} C_VEL
LIN {X 0,Y 591.97,Z 373.304,A -85,B 0,C 180,E1 28276.182,E2 28276.182} C_VEL
LIN {X 0,Y 591.962,Z 373.3,A -85,B 0,C 180,E1 28273.368,E2 28273.368} C_VEL
LIN {X 0,Y 591.99,Z 373.303,A -85,B 0,C 180,E1 28270.116,E2 28270.116} C_VEL
LIN {X 0,Y 591.957,Z 373.303,A -85,B 0,C 180,E1 28267.277,E2 28267.277} C_VEL
LIN {X 0,Y 592.031,Z 373.302,A -85,B 0,C 180,E1 28264.164,E2 28264.164} C_VEL
LIN {X 0,Y 591.957,Z 373.303,A -85,B 0,C 180,E1 28261.161,E2 28261.161} C_VEL
LIN {X 0,Y 592.024,Z 373.306,A -85,B 0,C 180,E1 28258.161,E2 28258.161} C_VEL
LIN {X 0,Y 591.961,Z 373.303,A -85,B 0,C 180,E1 28255.058,E2 28255.058} C_VEL
LIN {X 0,Y 591.984,Z 373.303,A -85,B 0,C 180,E1 28252.234,E2 28252.234} C_VEL
LIN {X 0,Y 591.977,Z 373.305,A -85,B 0,C 180,E1 28250.225,E2 28250.225} C_VEL
LIN {X 0,Y 591.035,Z 373.429,A -85,B 0,C 180,E1 28249.479,E2 28249.479} C_VEL
LIN {X 0,Y 584.496,Z 374.24,A -85,B 0,C 180,E1 28247.333,E2 28247.333} C_VEL
LIN {X 0,Y 584.032,Z 374.292,A -85,B 0,C 180,E1 28246.843,E2 28246.843} C_VEL
LIN {X 0,Y 584.035,Z 374.293,A -85,B 0,C 180,E1 28244,E2 28244} C_VEL
LIN {X 0,Y 584.035,Z 374.292,A -85,B 0,C 180,E1 28240.602,E2 28240.602} C_VEL
LIN {X 0,Y 584.034,Z 374.292,A -85,B 0,C 180,E1 28237.768,E2 28237.768} C_VEL
LIN {X 0,Y 584.045,Z 374.29,A -85,B 0,C 180,E1 28234.442,E2 28234.442} C_VEL
LIN {X 0,Y 584.032,Z 374.293,A -85,B 0,C 180,E1 28231.58,E2 28231.58} C_VEL
LIN {X 0,Y 584.058,Z 374.29,A -85,B 0,C 180,E1 28228.294,E2 28228.294} C_VEL
LIN {X 0,Y 584.029,Z 374.292,A -85,B 0,C 180,E1 28225.362,E2 28225.362} C_VEL
LIN {X 0,Y 584.069,Z 374.291,A -85,B 0,C 180,E1 28222.109,E2 28222.109} C_VEL
LIN {X 0,Y 584.027,Z 374.288,A -85,B 0,C 180,E1 28219.157,E2 28219.157} C_VEL
LIN {X 0,Y 584.088,Z 374.288,A -85,B 0,C 180,E1 28215.97,E2 28215.97} C_VEL
LIN {X 0,Y 584.027,Z 374.294,A -85,B 0,C 180,E1 28212.952,E2 28212.952} C_VEL
LIN {X 0,Y 584.1,Z 374.29,A -85,B 0,C 180,E1 28209.772,E2 28209.772} C_VEL
LIN {X 0,Y 584.028,Z 374.29,A -85,B 0,C 180,E1 28206.691,E2 28206.691} C_VEL
LIN {X 0,Y 584.106,Z 374.549,A -85,B 0,C 180,E1 28205.351,E2 28205.351} C_VEL
LIN {X 0,Y 585.694,Z 379.022,A -85,B 0,C 180,E1 28204.882,E2 28204.882} C_VEL
LIN {X 0,Y 586.934,Z 382.464,A -85,B 0,C 180,E1 28204.561,E2 28204.561} C_VEL
LIN {X 0,Y 586.419,Z 426.376,A -85,B 0,C 180,E1 28201.621,E2 28201.621} C_VEL
LIN {X 0,Y 586.077,Z 470.389,A -85,B 0,C 180,E1 28198.769,E2 28198.769} C_VEL
LIN {X 0,Y 586.688,Z 475.921,A -85,B 0,C 180,E1 28198.656,E2 28198.656} C_VEL
LIN {X 0,Y 586.074,Z 732.094,A -85,B 0,C 180,E1 28195.211,E2 28195.211} C_VEL
LIN {X 0,Y 585.921,Z 752.341,A -85,B 0,C 180,E1 28194.758,E2 28194.758} C_VEL
LIN {X 0,Y 585.734,Z 772.273,A -85,B 0,C 180,E1 28194.132,E2 28194.132} C_VEL
LIN {X 0,Y 585.506,Z 791.661,A -85,B 0,C 180,E1 28193.34,E2 28193.34} C_VEL
LIN {X 0,Y 585.3,Z 810.281,A -85,B 0,C 180,E1 28192.393,E2 28192.393} C_VEL
LIN {X 0,Y 585.055,Z 828.874,A -85,B 0,C 180,E1 28191.242,E2 28191.242} C_VEL
LIN {X 0,Y 584.803,Z 846.342,A -85,B 0,C 180,E1 28189.944,E2 28189.944} C_VEL
LIN {X 0,Y 584.581,Z 862.228,A -85,B 0,C 180,E1 28188.55,E2 28188.55} C_VEL
LIN {X 0,Y 584.391,Z 877.187,A -85,B 0,C 180,E1 28187.012,E2 28187.012} C_VEL
LIN {X 0,Y 584.234,Z 890.696,A -85,B 0,C 180,E1 28185.383,E2 28185.383} C_VEL
LIN {X 0,Y 584.113,Z 902.812,A -85,B 0,C 180,E1 28183.664,E2 28183.664} C_VEL
LIN {X 0,Y 584.025,Z 913.539,A -85,B 0,C 180,E1 28181.855,E2 28181.855} C_VEL
LIN {X 0,Y 583.964,Z 922.81,A -85,B 0,C 180,E1 28179.958,E2 28179.958} C_VEL
LIN {X 0,Y 583.934,Z 930.167,A -85,B 0,C 180,E1 28178.071,E2 28178.071} C_VEL
LIN {X 0,Y 583.921,Z 936.127,A -85,B 0,C 180,E1 28176.094,E2 28176.094} C_VEL
LIN {X 0,Y 583.917,Z 940.537,A -85,B 0,C 180,E1 28174.026,E2 28174.026} C_VEL
LIN {X 0,Y 583.916,Z 943.074,A -85,B 0,C 180,E1 28172.061,E2 28172.061} C_VEL
LIN {X 0,Y 583.913,Z 943.996,A -85,B 0,C 180,E1 28170,E2 28170} C_VEL
LIN {X 0,Y 583.916,Z 943.137,A -85,B 0,C 180,E1 28167.939,E2 28167.939} C_VEL
LIN {X 0,Y 583.918,Z 940.682,A -85,B 0,C 180,E1 28165.974,E2 28165.974} C_VEL
LIN {X 0,Y 583.923,Z 936.358,A -85,B 0,C 180,E1 28163.906,E2 28163.906} C_VEL
LIN {X 0,Y 583.937,Z 930.487,A -85,B 0,C 180,E1 28161.929,E2 28161.929} C_VEL
LIN {X 0,Y 583.962,Z 923.21,A -85,B 0,C 180,E1 28160.042,E2 28160.042} C_VEL
LIN {X 0,Y 584.017,Z 914.004,A -85,B 0,C 180,E1 28158.144,E2 28158.144} C_VEL
LIN {X 0,Y 584.103,Z 903.382,A -85,B 0,C 180,E1 28156.336,E2 28156.336} C_VEL
LIN {X 0,Y 584.228,Z 891.381,A -85,B 0,C 180,E1 28154.617,E2 28154.617} C_VEL
LIN {X 0,Y 584.386,Z 878,A -85,B 0,C 180,E1 28152.988,E2 28152.988} C_VEL
LIN {X 0,Y 584.576,Z 863.192,A -85,B 0,C 180,E1 28151.45,E2 28151.45} C_VEL
LIN {X 0,Y 584.801,Z 846.825,A -85,B 0,C 180,E1 28150.004,E2 28150.004} C_VEL
LIN {X 0,Y 585.049,Z 829.341,A -85,B 0,C 180,E1 28148.7,E2 28148.7} C_VEL
LIN {X 0,Y 585.287,Z 810.822,A -85,B 0,C 180,E1 28147.549,E2 28147.549} C_VEL
LIN {X 0,Y 585.499,Z 792.44,A -85,B 0,C 180,E1 28146.606,E2 28146.606} C_VEL
LIN {X 0,Y 585.73,Z 772.468,A -85,B 0,C 180,E1 28145.785,E2 28145.785} C_VEL
LIN {X 0,Y 585.921,Z 752.323,A -85,B 0,C 180,E1 28145.151,E2 28145.151} C_VEL
LIN {X 0,Y 586.073,Z 732.171,A -85,B 0,C 180,E1 28144.7,E2 28144.7} C_VEL
LIN {X 0,Y 586.676,Z 478.507,A -85,B 0,C 180,E1 28141.289,E2 28141.289} C_VEL
LIN {X 0,Y 586.392,Z 472.321,A -85,B 0,C 180,E1 28141.189,E2 28141.189} C_VEL
LIN {X 0,Y 586.027,Z 469.154,A -85,B 0,C 180,E1 28141.076,E2 28141.076} C_VEL
LIN {X 0,Y 586.491,Z 421.695,A -85,B 0,C 180,E1 28137.981,E2 28137.981} C_VEL
LIN {X 0,Y 586.938,Z 382.049,A -85,B 0,C 180,E1 28135.321,E2 28135.321} C_VEL
LIN {X 0,Y 584.138,Z 374.695,A -85,B 0,C 180,E1 28134.591,E2 28134.591} C_VEL
LIN {X 0,Y 584.093,Z 374.294,A -85,B 0,C 180,E1 28134.044,E2 28134.044} C_VEL
LIN {X 0,Y 584.037,Z 374.294,A -85,B 0,C 180,E1 28130.949,E2 28130.949} C_VEL
LIN {X 0,Y 584.087,Z 374.295,A -85,B 0,C 180,E1 28127.69,E2 28127.69} C_VEL
LIN {X 0,Y 584.035,Z 374.289,A -85,B 0,C 180,E1 28124.719,E2 28124.719} C_VEL
LIN {X 0,Y 584.096,Z 374.287,A -85,B 0,C 180,E1 28121.577,E2 28121.577} C_VEL
LIN {X 0,Y 584.032,Z 374.292,A -85,B 0,C 180,E1 28118.52,E2 28118.52} C_VEL
LIN {X 0,Y 584.097,Z 374.285,A -85,B 0,C 180,E1 28115.352,E2 28115.352} C_VEL
LIN {X 0,Y 584.03,Z 374.291,A -85,B 0,C 180,E1 28112.249,E2 28112.249} C_VEL
LIN {X 0,Y 584.098,Z 374.285,A -85,B 0,C 180,E1 28109.088,E2 28109.088} C_VEL
LIN {X 0,Y 584.029,Z 374.291,A -85,B 0,C 180,E1 28105.994,E2 28105.994} C_VEL
LIN {X 0,Y 584.099,Z 374.293,A -85,B 0,C 180,E1 28102.866,E2 28102.866} C_VEL
LIN {X 0,Y 584.027,Z 374.292,A -85,B 0,C 180,E1 28099.815,E2 28099.815} C_VEL
LIN {X 0,Y 584.098,Z 374.29,A -85,B 0,C 180,E1 28096.714,E2 28096.714} C_VEL
LIN {X 0,Y 584.026,Z 374.293,A -85,B 0,C 180,E1 28093.565,E2 28093.565} C_VEL
LIN {X 0,Y 584.085,Z 374.288,A -85,B 0,C 180,E1 28090.555,E2 28090.555} C_VEL
LIN {X 0,Y 584.025,Z 374.291,A -85,B 0,C 180,E1 28087.377,E2 28087.377} C_VEL
LIN {X 0,Y 584.067,Z 374.291,A -85,B 0,C 180,E1 28084.418,E2 28084.418} C_VEL
LIN {X 0,Y 584.028,Z 374.293,A -85,B 0,C 180,E1 28081.177,E2 28081.177} C_VEL
LIN {X 0,Y 584.045,Z 374.291,A -85,B 0,C 180,E1 28078.333,E2 28078.333} C_VEL
LIN {X 0,Y 584.03,Z 374.294,A -85,B 0,C 180,E1 28074.991,E2 28074.991} C_VEL
LIN {X 0,Y 584.038,Z 374.29,A -85,B 0,C 180,E1 28072.128,E2 28072.128} C_VEL
LIN {X 0,Y 584.029,Z 374.29,A -85,B 0,C 180,E1 28068.746,E2 28068.746} C_VEL
LIN {X 0,Y 584.031,Z 374.286,A -85,B 0,C 180,E1 28065.931,E2 28065.931} C_VEL
LIN {X 0,Y 584.034,Z 374.292,A -85,B 0,C 180,E1 28062.567,E2 28062.567} C_VEL
LIN {X 0,Y 584.024,Z 374.286,A -85,B 0,C 180,E1 28059.75,E2 28059.75} C_VEL
LIN {X 0,Y 584.051,Z 374.292,A -85,B 0,C 180,E1 28056.492,E2 28056.492} C_VEL
LIN {X 0,Y 584.019,Z 374.289,A -85,B 0,C 180,E1 28053.56,E2 28053.56} C_VEL
LIN {X 0,Y 584.065,Z 374.288,A -85,B 0,C 180,E1 28050.348,E2 28050.348} C_VEL
LIN {X 0,Y 584.015,Z 374.294,A -85,B 0,C 180,E1 28047.365,E2 28047.365} C_VEL
LIN {X 0,Y 584.086,Z 374.288,A -85,B 0,C 180,E1 28044.235,E2 28044.235} C_VEL
LIN {X 0,Y 584.011,Z 374.291,A -85,B 0,C 180,E1 28041.2,E2 28041.2} C_VEL
LIN {X 0,Y 584.092,Z 374.287,A -85,B 0,C 180,E1 28038.118,E2 28038.118} C_VEL
LIN {X 0,Y 584.011,Z 374.298,A -85,B 0,C 180,E1 28034.998,E2 28034.998} C_VEL
LIN {X 0,Y 584.107,Z 374.506,A -85,B 0,C 180,E1 28034.093,E2 28034.093} C_VEL
LIN {X 0,Y 584.607,Z 376.259,A -85,B 0,C 180,E1 28033.872,E2 28033.872} C_VEL
LIN {X 0,Y 586.758,Z 380.213,A -85,B 0,C 180,E1 28033.455,E2 28033.455} C_VEL
LIN {X 0,Y 589.163,Z 384.684,A -85,B 0,C 180,E1 28032.993,E2 28032.993} C_VEL
LIN {X 0,Y 588.516,Z 441.086,A -85,B 0,C 180,E1 28030.084,E2 28030.084} C_VEL
LIN {X 0,Y 588.42,Z 466.344,A -85,B 0,C 180,E1 28028.84,E2 28028.84} C_VEL
LIN {X 0,Y 588.91,Z 471.918,A -85,B 0,C 180,E1 28028.716,E2 28028.716} C_VEL
LIN {X 0,Y 588.197,Z 676.771,A -85,B 0,C 180,E1 28025.694,E2 28025.694} C_VEL
LIN {X 0,Y 587.71,Z 815.541,A -85,B 0,C 180,E1 28023.677,E2 28023.677} C_VEL
LIN {X 0,Y 587.465,Z 839.286,A -85,B 0,C 180,E1 28023.148,E2 28023.148} C_VEL
LIN {X 0,Y 587.254,Z 859.782,A -85,B 0,C 180,E1 28022.524,E2 28022.524} C_VEL
LIN {X 0,Y 586.874,Z 883.124,A -85,B 0,C 180,E1 28021.618,E2 28021.618} C_VEL
LIN {X 0,Y 586.588,Z 904.558,A -85,B 0,C 180,E1 28020.596,E2 28020.596} C_VEL
LIN {X 0,Y 586.172,Z 925.032,A -85,B 0,C 180,E1 28019.423,E2 28019.423} C_VEL
LIN {X 0,Y 585.85,Z 945.326,A -85,B 0,C 180,E1 28018.073,E2 28018.073} C_VEL
LIN {X 0,Y 585.465,Z 963.918,A -85,B 0,C 180,E1 28016.635,E2 28016.635} C_VEL
LIN {X 0,Y 585.12,Z 983.124,A -85,B 0,C 180,E1 28014.934,E2 28014.934} C_VEL
LIN {X 0,Y 584.853,Z 1000.156,A -85,B 0,C 180,E1 28013.209,E2 28013.209} C_VEL
LIN {X 0,Y 584.586,Z 1015.989,A -85,B 0,C 180,E1 28011.365,E2 28011.365} C_VEL
LIN {X 0,Y 584.38,Z 1030.912,A -85,B 0,C 180,E1 28009.386,E2 28009.386} C_VEL
LIN {X 0,Y 584.228,Z 1043.736,A -85,B 0,C 180,E1 28007.428,E2 28007.428} C_VEL
LIN {X 0,Y 584.091,Z 1055.793,A -85,B 0,C 180,E1 28005.285,E2 28005.285} C_VEL
LIN {X 0,Y 584,Z 1065.54,A -85,B 0,C 180,E1 28003.263,E2 28003.263} C_VEL
LIN {X 0,Y 583.944,Z 1074.337,A -85,B 0,C 180,E1 28001.056,E2 28001.056} C_VEL
LIN {X 0,Y 583.939,Z 1081.173,A -85,B 0,C 180,E1 27998.964,E2 27998.964} C_VEL
LIN {X 0,Y 583.905,Z 1086.84,A -85,B 0,C 180,E1 27996.687,E2 27996.687} C_VEL
LIN {X 0,Y 583.901,Z 1090.594,A -85,B 0,C 180,E1 27994.616,E2 27994.616} C_VEL
LIN {X 0,Y 583.915,Z 1093.055,A -85,B 0,C 180,E1 27992.355,E2 27992.355} C_VEL
LIN {X 0,Y 583.893,Z 1093.939,A -85,B 0,C 180,E1 27990.294,E2 27990.294} C_VEL
LIN {X 0,Y 583.91,Z 1093.323,A -85,B 0,C 180,E1 27988.037,E2 27988.037} C_VEL
LIN {X 0,Y 583.917,Z 1091.277,A -85,B 0,C 180,E1 27985.876,E2 27985.876} C_VEL
LIN {X 0,Y 583.923,Z 1087.46,A -85,B 0,C 180,E1 27983.61,E2 27983.61} C_VEL
LIN {X 0,Y 583.931,Z 1082.549,A -85,B 0,C 180,E1 27981.532,E2 27981.532} C_VEL
LIN {X 0,Y 583.948,Z 1075.406,A -85,B 0,C 180,E1 27979.243,E2 27979.243} C_VEL
LIN {X 0,Y 584.007,Z 1067.696,A -85,B 0,C 180,E1 27977.241,E2 27977.241} C_VEL
LIN {X 0,Y 584.086,Z 1057.357,A -85,B 0,C 180,E1 27975.02,E2 27975.02} C_VEL
LIN {X 0,Y 584.205,Z 1046.233,A -85,B 0,C 180,E1 27972.982,E2 27972.982} C_VEL
LIN {X 0,Y 584.345,Z 1033.038,A -85,B 0,C 180,E1 27970.924,E2 27970.924} C_VEL
LIN {X 0,Y 584.562,Z 1018.54,A -85,B 0,C 180,E1 27968.949,E2 27968.949} C_VEL
LIN {X 0,Y 584.782,Z 1003.432,A -85,B 0,C 180,E1 27967.157,E2 27967.157} C_VEL
LIN {X 0,Y 585.066,Z 985.673,A -85,B 0,C 180,E1 27965.312,E2 27965.312} C_VEL
LIN {X 0,Y 585.425,Z 968.25,A -85,B 0,C 180,E1 27963.721,E2 27963.721} C_VEL
LIN {X 0,Y 585.732,Z 949.33,A -85,B 0,C 180,E1 27962.224,E2 27962.224} C_VEL
LIN {X 0,Y 586.144,Z 927.701,A -85,B 0,C 180,E1 27960.743,E2 27960.743} C_VEL
LIN {X 0,Y 586.504,Z 907.833,A -85,B 0,C 180,E1 27959.581,E2 27959.581} C_VEL
LIN {X 0,Y 586.849,Z 886.215,A -85,B 0,C 180,E1 27958.519,E2 27958.519} C_VEL
LIN {X 0,Y 587.154,Z 865.509,A -85,B 0,C 180,E1 27957.676,E2 27957.676} C_VEL
LIN {X 0,Y 587.441,Z 842.856,A -85,B 0,C 180,E1 27956.951,E2 27956.951} C_VEL
LIN {X 0,Y 587.627,Z 821.764,A -85,B 0,C 180,E1 27956.438,E2 27956.438} C_VEL
LIN {X 0,Y 587.82,Z 790.551,A -85,B 0,C 180,E1 27955.94,E2 27955.94} C_VEL
LIN {X 0,Y 588.524,Z 580.703,A -85,B 0,C 180,E1 27952.902,E2 27952.902} C_VEL
LIN {X 0,Y 588.731,Z 468.475,A -85,B 0,C 180,E1 27951.217,E2 27951.217} C_VEL
LIN {X 0,Y 588.291,Z 463.341,A -85,B 0,C 180,E1 27951.034,E2 27951.034} C_VEL
LIN {X 0,Y 588.946,Z 403.994,A -85,B 0,C 180,E1 27948.018,E2 27948.018} C_VEL
LIN {X 0,Y 589.163,Z 384.684,A -85,B 0,C 180,E1 27947.007,E2 27947.007} C_VEL
LIN {X 0,Y 585.823,Z 378.366,A -85,B 0,C 180,E1 27946.357,E2 27946.357} C_VEL
LIN {X 0,Y 584.153,Z 374.73,A -85,B 0,C 180,E1 27945.962,E2 27945.962} C_VEL
LIN {X 0,Y 584.046,Z 374.269,A -85,B 0,C 180,E1 27945.691,E2 27945.691} C_VEL
LIN {X 0,Y 584.011,Z 374.285,A -85,B 0,C 180,E1 27942.819,E2 27942.819} C_VEL
LIN {X 0,Y 584.085,Z 374.286,A -85,B 0,C 180,E1 27939.681,E2 27939.681} C_VEL
LIN {X 0,Y 584.011,Z 374.295,A -85,B 0,C 180,E1 27936.691,E2 27936.691} C_VEL
LIN {X 0,Y 584.082,Z 374.292,A -85,B 0,C 180,E1 27933.685,E2 27933.685} C_VEL
LIN {X 0,Y 584.014,Z 374.288,A -85,B 0,C 180,E1 27930.552,E2 27930.552} C_VEL
LIN {X 0,Y 584.043,Z 374.295,A -85,B 0,C 180,E1 27927.737,E2 27927.737} C_VEL
LIN {X 0,Y 584.024,Z 374.291,A -85,B 0,C 180,E1 27924.475,E2 27924.475} C_VEL
LIN {X 0,Y 584.024,Z 374.294,A -85,B 0,C 180,E1 27921.703,E2 27921.703} C_VEL
LIN {X 0,Y 584.037,Z 374.291,A -85,B 0,C 180,E1 27918.361,E2 27918.361} C_VEL
LIN {X 0,Y 584.022,Z 374.294,A -85,B 0,C 180,E1 27915.49,E2 27915.49} C_VEL
LIN {X 0,Y 584.056,Z 374.288,A -85,B 0,C 180,E1 27912.256,E2 27912.256} C_VEL
LIN {X 0,Y 584.019,Z 374.293,A -85,B 0,C 180,E1 27909.36,E2 27909.36} C_VEL
LIN {X 0,Y 584.086,Z 374.291,A -85,B 0,C 180,E1 27906.191,E2 27906.191} C_VEL
LIN {X 0,Y 584.019,Z 374.292,A -85,B 0,C 180,E1 27903.14,E2 27903.14} C_VEL
LIN {X 0,Y 584.094,Z 374.292,A -85,B 0,C 180,E1 27900,E2 27900} C_VEL
LIN {X 0,Y 584.019,Z 374.292,A -85,B 0,C 180,E1 27896.957,E2 27896.957} C_VEL
LIN {X 0,Y 584.096,Z 374.294,A -85,B 0,C 180,E1 27893.907,E2 27893.907} C_VEL
LIN {X 0,Y 584.022,Z 374.293,A -85,B 0,C 180,E1 27890.838,E2 27890.838} C_VEL
LIN {X 0,Y 584.069,Z 374.292,A -85,B 0,C 180,E1 27887.844,E2 27887.844} C_VEL
LIN {X 0,Y 584.032,Z 374.292,A -85,B 0,C 180,E1 27886.843,E2 27886.843} C_VEL
LIN {X 0,Y 583.018,Z 374.421,A -85,B 0,C 180,E1 27886.087,E2 27886.087} C_VEL
LIN {X 0,Y 576.66,Z 375.222,A -85,B 0,C 180,E1 27883.966,E2 27883.966} C_VEL
LIN {X 0,Y 576.159,Z 375.282,A -85,B 0,C 180,E1 27883.414,E2 27883.414} C_VEL
LIN {X 0,Y 576.084,Z 375.281,A -85,B 0,C 180,E1 27880.323,E2 27880.323} C_VEL
LIN {X 0,Y 576.139,Z 375.281,A -85,B 0,C 180,E1 27877.339,E2 27877.339} C_VEL
LIN {X 0,Y 576.089,Z 375.28,A -85,B 0,C 180,E1 27874.174,E2 27874.174} C_VEL
LIN {X 0,Y 576.122,Z 375.283,A -85,B 0,C 180,E1 27871.215,E2 27871.215} C_VEL
LIN {X 0,Y 576.092,Z 375.28,A -85,B 0,C 180,E1 27867.921,E2 27867.921} C_VEL
LIN {X 0,Y 576.121,Z 375.282,A -85,B 0,C 180,E1 27864.939,E2 27864.939} C_VEL
LIN {X 0,Y 576.093,Z 375.282,A -85,B 0,C 180,E1 27861.674,E2 27861.674} C_VEL
LIN {X 0,Y 576.117,Z 375.275,A -85,B 0,C 180,E1 27858.719,E2 27858.719} C_VEL
LIN {X 0,Y 576.098,Z 375.277,A -85,B 0,C 180,E1 27855.479,E2 27855.479} C_VEL
LIN {X 0,Y 576.105,Z 375.284,A -85,B 0,C 180,E1 27852.6,E2 27852.6} C_VEL
LIN {X 0,Y 576.106,Z 375.285,A -85,B 0,C 180,E1 27849.28,E2 27849.28} C_VEL
LIN {X 0,Y 576.104,Z 375.279,A -85,B 0,C 180,E1 27846.361,E2 27846.361} C_VEL
LIN {X 0,Y 576.211,Z 375.636,A -85,B 0,C 180,E1 27845.822,E2 27845.822} C_VEL
LIN {X 0,Y 579.937,Z 385.187,A -85,B 0,C 180,E1 27844.848,E2 27844.848} C_VEL
LIN {X 0,Y 579.317,Z 427.248,A -85,B 0,C 180,E1 27841.996,E2 27841.996} C_VEL
LIN {X 0,Y 578.856,Z 470.503,A -85,B 0,C 180,E1 27839.161,E2 27839.161} C_VEL
LIN {X 0,Y 579.666,Z 477.042,A -85,B 0,C 180,E1 27839.021,E2 27839.021} C_VEL
LIN {X 0,Y 578.833,Z 732.029,A -85,B 0,C 180,E1 27835.551,E2 27835.551} C_VEL
LIN {X 0,Y 578.63,Z 752.27,A -85,B 0,C 180,E1 27835.094,E2 27835.094} C_VEL
LIN {X 0,Y 578.375,Z 772.294,A -85,B 0,C 180,E1 27834.459,E2 27834.459} C_VEL
LIN {X 0,Y 578.086,Z 791.673,A -85,B 0,C 180,E1 27833.658,E2 27833.658} C_VEL
LIN {X 0,Y 577.794,Z 810.29,A -85,B 0,C 180,E1 27832.7,E2 27832.7} C_VEL
LIN {X 0,Y 577.46,Z 828.885,A -85,B 0,C 180,E1 27831.535,E2 27831.535} C_VEL
LIN {X 0,Y 577.123,Z 846.14,A -85,B 0,C 180,E1 27830.238,E2 27830.238} C_VEL
LIN {X 0,Y 576.823,Z 862.235,A -85,B 0,C 180,E1 27828.809,E2 27828.809} C_VEL
LIN {X 0,Y 576.567,Z 877.193,A -85,B 0,C 180,E1 27827.25,E2 27827.25} C_VEL
LIN {X 0,Y 576.353,Z 890.702,A -85,B 0,C 180,E1 27825.599,E2 27825.599} C_VEL
LIN {X 0,Y 576.183,Z 903.457,A -85,B 0,C 180,E1 27823.753,E2 27823.753} C_VEL
LIN {X 0,Y 576.065,Z 914.062,A -85,B 0,C 180,E1 27821.92,E2 27821.92} C_VEL
LIN {X 0,Y 575.985,Z 923.254,A -85,B 0,C 180,E1 27819.997,E2 27819.997} C_VEL
LIN {X 0,Y 575.941,Z 930.875,A -85,B 0,C 180,E1 27817.983,E2 27817.983} C_VEL
LIN {X 0,Y 575.924,Z 936.382,A -85,B 0,C 180,E1 27816.079,E2 27816.079} C_VEL
LIN {X 0,Y 575.917,Z 940.697,A -85,B 0,C 180,E1 27813.982,E2 27813.982} C_VEL
LIN {X 0,Y 575.916,Z 943.142,A -85,B 0,C 180,E1 27811.99,E2 27811.99} C_VEL
LIN {X 0,Y 575.914,Z 943.994,A -85,B 0,C 180,E1 27809.901,E2 27809.901} C_VEL
LIN {X 0,Y 575.912,Z 943.068,A -85,B 0,C 180,E1 27807.811,E2 27807.811} C_VEL
LIN {X 0,Y 575.919,Z 940.523,A -85,B 0,C 180,E1 27805.818,E2 27805.818} C_VEL
LIN {X 0,Y 575.928,Z 936.356,A -85,B 0,C 180,E1 27803.821,E2 27803.821} C_VEL
LIN {X 0,Y 575.947,Z 930.485,A -85,B 0,C 180,E1 27801.816,E2 27801.816} C_VEL
LIN {X 0,Y 575.987,Z 922.853,A -85,B 0,C 180,E1 27799.821,E2 27799.821} C_VEL
LIN {X 0,Y 576.077,Z 913.484,A -85,B 0,C 180,E1 27797.877,E2 27797.877} C_VEL
LIN {X 0,Y 576.195,Z 902.739,A -85,B 0,C 180,E1 27796.042,E2 27796.042} C_VEL
LIN {X 0,Y 576.354,Z 890.601,A -85,B 0,C 180,E1 27794.298,E2 27794.298} C_VEL
LIN {X 0,Y 576.567,Z 877.066,A -85,B 0,C 180,E1 27792.646,E2 27792.646} C_VEL
LIN {X 0,Y 576.825,Z 862.081,A -85,B 0,C 180,E1 27791.086,E2 27791.086} C_VEL
LIN {X 0,Y 577.125,Z 846.159,A -85,B 0,C 180,E1 27789.674,E2 27789.674} C_VEL
LIN {X 0,Y 577.464,Z 828.641,A -85,B 0,C 180,E1 27788.358,E2 27788.358} C_VEL
LIN {X 0,Y 577.798,Z 809.992,A -85,B 0,C 180,E1 27787.193,E2 27787.193} C_VEL
LIN {X 0,Y 578.098,Z 791.296,A -85,B 0,C 180,E1 27786.235,E2 27786.235} C_VEL
LIN {X 0,Y 578.372,Z 772.218,A -85,B 0,C 180,E1 27785.448,E2 27785.448} C_VEL
LIN {X 0,Y 578.633,Z 751.779,A -85,B 0,C 180,E1 27784.803,E2 27784.803} C_VEL
LIN {X 0,Y 578.834,Z 731.623,A -85,B 0,C 180,E1 27784.353,E2 27784.353} C_VEL
LIN {X 0,Y 579.658,Z 477.275,A -85,B 0,C 180,E1 27780.892,E2 27780.892} C_VEL
LIN {X 0,Y 579.047,Z 471.728,A -85,B 0,C 180,E1 27780.781,E2 27780.781} C_VEL
LIN {X 0,Y 578.797,Z 469.085,A -85,B 0,C 180,E1 27780.676,E2 27780.676} C_VEL
LIN {X 0,Y 579.426,Z 421.684,A -85,B 0,C 180,E1 27777.543,E2 27777.543} C_VEL
LIN {X 0,Y 579.862,Z 385.012,A -85,B 0,C 180,E1 27775.044,E2 27775.044} C_VEL
LIN {X 0,Y 576.211,Z 375.651,A -85,B 0,C 180,E1 27774.09,E2 27774.09} C_VEL
LIN {X 0,Y 576.098,Z 375.276,A -85,B 0,C 180,E1 27773.306,E2 27773.306} C_VEL
LIN {X 0,Y 576.164,Z 375.277,A -85,B 0,C 180,E1 27770.181,E2 27770.181} C_VEL
LIN {X 0,Y 576.096,Z 375.282,A -85,B 0,C 180,E1 27766.944,E2 27766.944} C_VEL
LIN {X 0,Y 576.163,Z 375.277,A -85,B 0,C 180,E1 27763.787,E2 27763.787} C_VEL
LIN {X 0,Y 576.093,Z 375.275,A -85,B 0,C 180,E1 27760.606,E2 27760.606} C_VEL
LIN {X 0,Y 576.163,Z 375.281,A -85,B 0,C 180,E1 27757.526,E2 27757.526} C_VEL
LIN {X 0,Y 576.092,Z 375.28,A -85,B 0,C 180,E1 27754.338,E2 27754.338} C_VEL
LIN {X 0,Y 576.157,Z 375.273,A -85,B 0,C 180,E1 27751.141,E2 27751.141} C_VEL
LIN {X 0,Y 576.09,Z 375.28,A -85,B 0,C 180,E1 27748.057,E2 27748.057} C_VEL
LIN {X 0,Y 576.16,Z 375.279,A -85,B 0,C 180,E1 27744.942,E2 27744.942} C_VEL
LIN {X 0,Y 576.089,Z 375.279,A -85,B 0,C 180,E1 27741.79,E2 27741.79} C_VEL
LIN {X 0,Y 576.158,Z 375.28,A -85,B 0,C 180,E1 27738.622,E2 27738.622} C_VEL
LIN {X 0,Y 576.087,Z 375.28,A -85,B 0,C 180,E1 27735.503,E2 27735.503} C_VEL
LIN {X 0,Y 576.158,Z 375.281,A -85,B 0,C 180,E1 27732.303,E2 27732.303} C_VEL
LIN {X 0,Y 576.087,Z 375.281,A -85,B 0,C 180,E1 27729.188,E2 27729.188} C_VEL
LIN {X 0,Y 576.158,Z 375.281,A -85,B 0,C 180,E1 27726.074,E2 27726.074} C_VEL
LIN {X 0,Y 576.084,Z 375.28,A -85,B 0,C 180,E1 27722.985,E2 27722.985} C_VEL
LIN {X 0,Y 576.155,Z 375.28,A -85,B 0,C 180,E1 27719.801,E2 27719.801} C_VEL
LIN {X 0,Y 576.082,Z 375.281,A -85,B 0,C 180,E1 27716.717,E2 27716.717} C_VEL
LIN {X 0,Y 576.16,Z 375.282,A -85,B 0,C 180,E1 27713.524,E2 27713.524} C_VEL
LIN {X 0,Y 576.081,Z 375.282,A -85,B 0,C 180,E1 27710.409,E2 27710.409} C_VEL
LIN {X 0,Y 576.154,Z 375.27,A -85,B 0,C 180,E1 27707.24,E2 27707.24} C_VEL
LIN {X 0,Y 576.08,Z 375.282,A -85,B 0,C 180,E1 27704.188,E2 27704.188} C_VEL
LIN {X 0,Y 576.156,Z 375.272,A -85,B 0,C 180,E1 27701.049,E2 27701.049} C_VEL
LIN {X 0,Y 576.078,Z 375.283,A -85,B 0,C 180,E1 27697.947,E2 27697.947} C_VEL
LIN {X 0,Y 576.154,Z 375.273,A -85,B 0,C 180,E1 27694.839,E2 27694.839} C_VEL
LIN {X 0,Y 576.077,Z 375.284,A -85,B 0,C 180,E1 27691.717,E2 27691.717} C_VEL
LIN {X 0,Y 576.15,Z 375.272,A -85,B 0,C 180,E1 27688.626,E2 27688.626} C_VEL
LIN {X 0,Y 576.075,Z 375.279,A -85,B 0,C 180,E1 27685.531,E2 27685.531} C_VEL
LIN {X 0,Y 576.119,Z 375.284,A -85,B 0,C 180,E1 27682.597,E2 27682.597} C_VEL
LIN {X 0,Y 576.08,Z 375.287,A -85,B 0,C 180,E1 27679.394,E2 27679.394} C_VEL
LIN {X 0,Y 576.096,Z 375.272,A -85,B 0,C 180,E1 27676.508,E2 27676.508} C_VEL
LIN {X 0,Y 576.105,Z 375.512,A -85,B 0,C 180,E1 27674.8,E2 27674.8} C_VEL
LIN {X 0,Y 576.719,Z 377.544,A -85,B 0,C 180,E1 27674.558,E2 27674.558} C_VEL
LIN {X 0,Y 578.914,Z 381.165,A -85,B 0,C 180,E1 27674.142,E2 27674.142} C_VEL
LIN {X 0,Y 582.964,Z 388.639,A -85,B 0,C 180,E1 27673.347,E2 27673.347} C_VEL
LIN {X 0,Y 582.086,Z 444.794,A -85,B 0,C 180,E1 27670.424,E2 27670.424} C_VEL
LIN {X 0,Y 581.958,Z 466.341,A -85,B 0,C 180,E1 27669.355,E2 27669.355} C_VEL
LIN {X 0,Y 582.657,Z 472.935,A -85,B 0,C 180,E1 27669.195,E2 27669.195} C_VEL
LIN {X 0,Y 581.693,Z 677.789,A -85,B 0,C 180,E1 27666.141,E2 27666.141} C_VEL
LIN {X 0,Y 581.041,Z 815.756,A -85,B 0,C 180,E1 27664.113,E2 27664.113} C_VEL
LIN {X 0,Y 580.712,Z 839.591,A -85,B 0,C 180,E1 27663.575,E2 27663.575} C_VEL
LIN {X 0,Y 580.42,Z 860.7,A -85,B 0,C 180,E1 27662.924,E2 27662.924} C_VEL
LIN {X 0,Y 579.954,Z 882.402,A -85,B 0,C 180,E1 27662.073,E2 27662.073} C_VEL
LIN {X 0,Y 579.555,Z 902.543,A -85,B 0,C 180,E1 27661.112,E2 27661.112} C_VEL
LIN {X 0,Y 579.023,Z 924.145,A -85,B 0,C 180,E1 27659.88,E2 27659.88} C_VEL
LIN {X 0,Y 578.575,Z 944.186,A -85,B 0,C 180,E1 27658.544,E2 27658.544} C_VEL
LIN {X 0,Y 578.038,Z 963.682,A -85,B 0,C 180,E1 27657.025,E2 27657.025} C_VEL
LIN {X 0,Y 577.574,Z 983.349,A -85,B 0,C 180,E1 27655.26,E2 27655.26} C_VEL
LIN {X 0,Y 577.192,Z 1000.672,A -85,B 0,C 180,E1 27653.48,E2 27653.48} C_VEL
LIN {X 0,Y 576.821,Z 1016.842,A -85,B 0,C 180,E1 27651.56,E2 27651.56} C_VEL
LIN {X 0,Y 576.525,Z 1032.331,A -85,B 0,C 180,E1 27649.45,E2 27649.45} C_VEL
LIN {X 0,Y 576.328,Z 1045.334,A -85,B 0,C 180,E1 27647.412,E2 27647.412} C_VEL
LIN {X 0,Y 576.15,Z 1056.836,A -85,B 0,C 180,E1 27645.295,E2 27645.295} C_VEL
LIN {X 0,Y 576.037,Z 1066.879,A -85,B 0,C 180,E1 27643.143,E2 27643.143} C_VEL
LIN {X 0,Y 575.96,Z 1075.051,A -85,B 0,C 180,E1 27641.009,E2 27641.009} C_VEL
LIN {X 0,Y 575.939,Z 1082.04,A -85,B 0,C 180,E1 27638.788,E2 27638.788} C_VEL
LIN {X 0,Y 575.916,Z 1087.254,A -85,B 0,C 180,E1 27636.58,E2 27636.58} C_VEL
LIN {X 0,Y 575.913,Z 1091.163,A -85,B 0,C 180,E1 27634.281,E2 27634.281} C_VEL
LIN {X 0,Y 575.914,Z 1093.256,A -85,B 0,C 180,E1 27632.089,E2 27632.089} C_VEL
LIN {X 0,Y 575.899,Z 1093.962,A -85,B 0,C 180,E1 27629.801,E2 27629.801} C_VEL
LIN {X 0,Y 575.916,Z 1093.122,A -85,B 0,C 180,E1 27627.711,E2 27627.711} C_VEL
LIN {X 0,Y 575.902,Z 1090.753,A -85,B 0,C 180,E1 27625.419,E2 27625.419} C_VEL
LIN {X 0,Y 575.903,Z 1086.909,A -85,B 0,C 180,E1 27623.253,E2 27623.253} C_VEL
LIN {X 0,Y 575.947,Z 1081.475,A -85,B 0,C 180,E1 27621.011,E2 27621.011} C_VEL
LIN {X 0,Y 575.961,Z 1074.694,A -85,B 0,C 180,E1 27618.89,E2 27618.89} C_VEL
LIN {X 0,Y 576.037,Z 1066.456,A -85,B 0,C 180,E1 27616.755,E2 27616.755} C_VEL
LIN {X 0,Y 576.152,Z 1056.316,A -85,B 0,C 180,E1 27614.602,E2 27614.602} C_VEL
LIN {X 0,Y 576.337,Z 1044.375,A -85,B 0,C 180,E1 27612.43,E2 27612.43} C_VEL
LIN {X 0,Y 576.543,Z 1031.622,A -85,B 0,C 180,E1 27610.445,E2 27610.445} C_VEL
LIN {X 0,Y 576.821,Z 1016.842,A -85,B 0,C 180,E1 27608.44,E2 27608.44} C_VEL
LIN {X 0,Y 577.192,Z 1000.672,A -85,B 0,C 180,E1 27606.52,E2 27606.52} C_VEL
LIN {X 0,Y 577.574,Z 983.349,A -85,B 0,C 180,E1 27604.74,E2 27604.74} C_VEL
LIN {X 0,Y 578.038,Z 963.68,A -85,B 0,C 180,E1 27602.975,E2 27602.975} C_VEL
LIN {X 0,Y 578.573,Z 944.183,A -85,B 0,C 180,E1 27601.456,E2 27601.456} C_VEL
LIN {X 0,Y 579.038,Z 923.692,A -85,B 0,C 180,E1 27600.092,E2 27600.092} C_VEL
LIN {X 0,Y 579.565,Z 901.426,A -85,B 0,C 180,E1 27598.831,E2 27598.831} C_VEL
LIN {X 0,Y 580.001,Z 880.991,A -85,B 0,C 180,E1 27597.865,E2 27597.865} C_VEL
LIN {X 0,Y 580.44,Z 858.169,A -85,B 0,C 180,E1 27596.991,E2 27596.991} C_VEL
LIN {X 0,Y 580.75,Z 837.274,A -85,B 0,C 180,E1 27596.361,E2 27596.361} C_VEL
LIN {X 0,Y 581.05,Z 814.169,A -85,B 0,C 180,E1 27595.86,E2 27595.86} C_VEL
LIN {X 0,Y 582.108,Z 588.403,A -85,B 0,C 180,E1 27592.54,E2 27592.54} C_VEL
LIN {X 0,Y 582.494,Z 470.024,A -85,B 0,C 180,E1 27590.747,E2 27590.747} C_VEL
LIN {X 0,Y 581.828,Z 463.959,A -85,B 0,C 180,E1 27590.549,E2 27590.549} C_VEL
LIN {X 0,Y 582.71,Z 404.781,A -85,B 0,C 180,E1 27587.506,E2 27587.506} C_VEL
LIN {X 0,Y 582.964,Z 388.638,A -85,B 0,C 180,E1 27586.653,E2 27586.653} C_VEL
LIN {X 0,Y 578.232,Z 379.772,A -85,B 0,C 180,E1 27585.714,E2 27585.714} C_VEL
LIN {X 0,Y 576.325,Z 376.482,A -85,B 0,C 180,E1 27585.341,E2 27585.341} C_VEL
LIN {X 0,Y 576.081,Z 375.358,A -85,B 0,C 180,E1 27585.134,E2 27585.134} C_VEL
LIN {X 0,Y 576.122,Z 375.272,A -85,B 0,C 180,E1 27582.178,E2 27582.178} C_VEL
LIN {X 0,Y 576.075,Z 375.279,A -85,B 0,C 180,E1 27578.961,E2 27578.961} C_VEL
LIN {X 0,Y 576.096,Z 375.285,A -85,B 0,C 180,E1 27576.163,E2 27576.163} C_VEL
LIN {X 0,Y 576.086,Z 375.284,A -85,B 0,C 180,E1 27572.855,E2 27572.855} C_VEL
LIN {X 0,Y 576.088,Z 375.276,A -85,B 0,C 180,E1 27569.99,E2 27569.99} C_VEL
LIN {X 0,Y 576.088,Z 375.277,A -85,B 0,C 180,E1 27566.601,E2 27566.601} C_VEL
LIN {X 0,Y 576.088,Z 375.281,A -85,B 0,C 180,E1 27563.744,E2 27563.744} C_VEL
LIN {X 0,Y 576.087,Z 375.274,A -85,B 0,C 180,E1 27560.311,E2 27560.311} C_VEL
LIN {X 0,Y 576.089,Z 375.281,A -85,B 0,C 180,E1 27557.473,E2 27557.473} C_VEL
LIN {X 0,Y 576.09,Z 375.274,A -85,B 0,C 180,E1 27554.062,E2 27554.062} C_VEL
LIN {X 0,Y 576.09,Z 375.277,A -85,B 0,C 180,E1 27551.209,E2 27551.209} C_VEL
LIN {X 0,Y 576.09,Z 375.279,A -85,B 0,C 180,E1 27547.78,E2 27547.78} C_VEL
LIN {X 0,Y 576.089,Z 375.282,A -85,B 0,C 180,E1 27544.969,E2 27544.969} C_VEL
LIN {X 0,Y 576.099,Z 375.28,A -85,B 0,C 180,E1 27541.591,E2 27541.591} C_VEL
LIN {X 0,Y 576.09,Z 375.282,A -85,B 0,C 180,E1 27538.707,E2 27538.707} C_VEL
LIN {X 0,Y 576.1,Z 375.281,A -85,B 0,C 180,E1 27535.321,E2 27535.321} C_VEL
LIN {X 0,Y 576.085,Z 375.28,A -85,B 0,C 180,E1 27532.52,E2 27532.52} C_VEL
LIN {X 0,Y 576.126,Z 375.278,A -85,B 0,C 180,E1 27529.298,E2 27529.298} C_VEL
LIN {X 0,Y 576.084,Z 375.282,A -85,B 0,C 180,E1 27526.347,E2 27526.347} C_VEL
LIN {X 0,Y 576.159,Z 375.282,A -85,B 0,C 180,E1 27523.414,E2 27523.414} C_VEL
LIN {X 0,Y 575.182,Z 375.4,A -85,B 0,C 180,E1 27522.648,E2 27522.648} C_VEL
LIN {X 0,Y 568.676,Z 376.206,A -85,B 0,C 180,E1 27520.499,E2 27520.499} C_VEL
LIN {X 0,Y 568.152,Z 376.271,A -85,B 0,C 180,E1 27519.938,E2 27519.938} C_VEL
LIN {X 0,Y 568.181,Z 376.27,A -85,B 0,C 180,E1 27516.675,E2 27516.675} C_VEL
LIN {X 0,Y 568.153,Z 376.27,A -85,B 0,C 180,E1 27513.674,E2 27513.674} C_VEL
LIN {X 0,Y 568.175,Z 376.257,A -85,B 0,C 180,E1 27510.363,E2 27510.363} C_VEL
LIN {X 0,Y 568.153,Z 376.271,A -85,B 0,C 180,E1 27507.417,E2 27507.417} C_VEL
LIN {X 0,Y 568.182,Z 376.259,A -85,B 0,C 180,E1 27504.126,E2 27504.126} C_VEL
LIN {X 0,Y 568.151,Z 376.272,A -85,B 0,C 180,E1 27501.207,E2 27501.207} C_VEL
LIN {X 0,Y 568.197,Z 376.269,A -85,B 0,C 180,E1 27497.954,E2 27497.954} C_VEL
LIN {X 0,Y 568.153,Z 376.268,A -85,B 0,C 180,E1 27494.886,E2 27494.886} C_VEL
LIN {X 0,Y 568.183,Z 376.263,A -85,B 0,C 180,E1 27491.562,E2 27491.562} C_VEL
LIN {X 0,Y 568.159,Z 376.276,A -85,B 0,C 180,E1 27488.534,E2 27488.534} C_VEL
LIN {X 0,Y 568.19,Z 376.492,A -85,B 0,C 180,E1 27486.467,E2 27486.467} C_VEL
LIN {X 0,Y 569.231,Z 379.343,A -85,B 0,C 180,E1 27486.099,E2 27486.099} C_VEL
LIN {X 0,Y 572.999,Z 388.814,A -85,B 0,C 180,E1 27485.076,E2 27485.076} C_VEL
LIN {X 0,Y 572.15,Z 432.983,A -85,B 0,C 180,E1 27482.052,E2 27482.052} C_VEL
LIN {X 0,Y 571.675,Z 470.694,A -85,B 0,C 180,E1 27479.561,E2 27479.561} C_VEL
LIN {X 0,Y 572.668,Z 478.14,A -85,B 0,C 180,E1 27479.396,E2 27479.396} C_VEL
LIN {X 0,Y 571.613,Z 731.858,A -85,B 0,C 180,E1 27475.9,E2 27475.9} C_VEL
LIN {X 0,Y 571.36,Z 752.142,A -85,B 0,C 180,E1 27475.44,E2 27475.44} C_VEL
LIN {X 0,Y 571.036,Z 772.315,A -85,B 0,C 180,E1 27474.794,E2 27474.794} C_VEL
LIN {X 0,Y 570.661,Z 792.519,A -85,B 0,C 180,E1 27473.944,E2 27473.944} C_VEL
LIN {X 0,Y 570.283,Z 811.108,A -85,B 0,C 180,E1 27472.967,E2 27472.967} C_VEL
LIN {X 0,Y 569.881,Z 828.896,A -85,B 0,C 180,E1 27471.836,E2 27471.836} C_VEL
LIN {X 0,Y 569.454,Z 846.364,A -85,B 0,C 180,E1 27470.505,E2 27470.505} C_VEL
LIN {X 0,Y 569.074,Z 862.556,A -85,B 0,C 180,E1 27469.045,E2 27469.045} C_VEL
LIN {X 0,Y 568.757,Z 877.199,A -85,B 0,C 180,E1 27467.495,E2 27467.495} C_VEL
LIN {X 0,Y 568.483,Z 890.709,A -85,B 0,C 180,E1 27465.82,E2 27465.82} C_VEL
LIN {X 0,Y 568.266,Z 903.462,A -85,B 0,C 180,E1 27463.949,E2 27463.949} C_VEL
LIN {X 0,Y 568.116,Z 914.067,A -85,B 0,C 180,E1 27462.089,E2 27462.089} C_VEL
LIN {X 0,Y 568.01,Z 923.257,A -85,B 0,C 180,E1 27460.139,E2 27460.139} C_VEL
LIN {X 0,Y 567.952,Z 930.878,A -85,B 0,C 180,E1 27458.096,E2 27458.096} C_VEL
LIN {X 0,Y 567.929,Z 936.385,A -85,B 0,C 180,E1 27456.165,E2 27456.165} C_VEL
LIN {X 0,Y 567.918,Z 940.698,A -85,B 0,C 180,E1 27454.038,E2 27454.038} C_VEL
LIN {X 0,Y 567.916,Z 943.142,A -85,B 0,C 180,E1 27452.018,E2 27452.018} C_VEL
LIN {X 0,Y 567.914,Z 943.994,A -85,B 0,C 180,E1 27449.899,E2 27449.899} C_VEL
LIN {X 0,Y 567.912,Z 943.067,A -85,B 0,C 180,E1 27447.78,E2 27447.78} C_VEL
LIN {X 0,Y 567.918,Z 940.523,A -85,B 0,C 180,E1 27445.759,E2 27445.759} C_VEL
LIN {X 0,Y 567.932,Z 936.355,A -85,B 0,C 180,E1 27443.733,E2 27443.733} C_VEL
LIN {X 0,Y 567.959,Z 930.483,A -85,B 0,C 180,E1 27441.7,E2 27441.7} C_VEL
LIN {X 0,Y 568.012,Z 923.111,A -85,B 0,C 180,E1 27439.737,E2 27439.737} C_VEL
LIN {X 0,Y 568.118,Z 914,A -85,B 0,C 180,E1 27437.808,E2 27437.808} C_VEL
LIN {X 0,Y 568.268,Z 903.376,A -85,B 0,C 180,E1 27435.948,E2 27435.948} C_VEL
LIN {X 0,Y 568.471,Z 891.338,A -85,B 0,C 180,E1 27434.175,E2 27434.175} C_VEL
LIN {X 0,Y 568.738,Z 877.987,A -85,B 0,C 180,E1 27432.505,E2 27432.505} C_VEL
LIN {X 0,Y 569.063,Z 863.18,A -85,B 0,C 180,E1 27430.925,E2 27430.925} C_VEL
LIN {X 0,Y 569.45,Z 846.814,A -85,B 0,C 180,E1 27429.441,E2 27429.441} C_VEL
LIN {X 0,Y 569.87,Z 829.39,A -85,B 0,C 180,E1 27428.109,E2 27428.109} C_VEL
LIN {X 0,Y 570.287,Z 810.841,A -85,B 0,C 180,E1 27426.928,E2 27426.928} C_VEL
LIN {X 0,Y 570.667,Z 792.411,A -85,B 0,C 180,E1 27425.961,E2 27425.961} C_VEL
LIN {X 0,Y 571.032,Z 772.461,A -85,B 0,C 180,E1 27425.121,E2 27425.121} C_VEL
LIN {X 0,Y 571.361,Z 752.144,A -85,B 0,C 180,E1 27424.47,E2 27424.47} C_VEL
LIN {X 0,Y 571.613,Z 731.89,A -85,B 0,C 180,E1 27424.01,E2 27424.01} C_VEL
LIN {X 0,Y 572.649,Z 481.205,A -85,B 0,C 180,E1 27420.557,E2 27420.557} C_VEL
LIN {X 0,Y 572.374,Z 474.873,A -85,B 0,C 180,E1 27420.452,E2 27420.452} C_VEL
LIN {X 0,Y 571.6,Z 470.056,A -85,B 0,C 180,E1 27420.328,E2 27420.328} C_VEL
LIN {X 0,Y 572.369,Z 422.744,A -85,B 0,C 180,E1 27417.167,E2 27417.167} C_VEL
LIN {X 0,Y 572.925,Z 388.496,A -85,B 0,C 180,E1 27414.806,E2 27414.806} C_VEL
LIN {X 0,Y 569.375,Z 379.564,A -85,B 0,C 180,E1 27413.84,E2 27413.84} C_VEL
LIN {X 0,Y 568.191,Z 376.472,A -85,B 0,C 180,E1 27413.44,E2 27413.44} C_VEL
LIN {X 0,Y 568.184,Z 376.273,A -85,B 0,C 180,E1 27410.56,E2 27410.56} C_VEL
LIN {X 0,Y 568.165,Z 376.273,A -85,B 0,C 180,E1 27407.209,E2 27407.209} C_VEL
LIN {X 0,Y 568.2,Z 376.263,A -85,B 0,C 180,E1 27404.114,E2 27404.114} C_VEL
LIN {X 0,Y 568.159,Z 376.263,A -85,B 0,C 180,E1 27400.823,E2 27400.823} C_VEL
LIN {X 0,Y 568.224,Z 376.269,A -85,B 0,C 180,E1 27397.643,E2 27397.643} C_VEL
LIN {X 0,Y 568.153,Z 376.269,A -85,B 0,C 180,E1 27394.374,E2 27394.374} C_VEL
LIN {X 0,Y 568.222,Z 376.261,A -85,B 0,C 180,E1 27391.22,E2 27391.22} C_VEL
LIN {X 0,Y 568.152,Z 376.27,A -85,B 0,C 180,E1 27388.141,E2 27388.141} C_VEL
LIN {X 0,Y 568.221,Z 376.267,A -85,B 0,C 180,E1 27384.981,E2 27384.981} C_VEL
LIN {X 0,Y 568.15,Z 376.268,A -85,B 0,C 180,E1 27381.798,E2 27381.798} C_VEL
LIN {X 0,Y 568.217,Z 376.268,A -85,B 0,C 180,E1 27378.572,E2 27378.572} C_VEL
LIN {X 0,Y 568.148,Z 376.269,A -85,B 0,C 180,E1 27375.516,E2 27375.516} C_VEL
LIN {X 0,Y 568.223,Z 376.271,A -85,B 0,C 180,E1 27372.397,E2 27372.397} C_VEL
LIN {X 0,Y 568.148,Z 376.271,A -85,B 0,C 180,E1 27369.216,E2 27369.216} C_VEL
LIN {X 0,Y 568.218,Z 376.27,A -85,B 0,C 180,E1 27366.061,E2 27366.061} C_VEL
LIN {X 0,Y 568.146,Z 376.269,A -85,B 0,C 180,E1 27362.926,E2 27362.926} C_VEL
LIN {X 0,Y 568.206,Z 376.269,A -85,B 0,C 180,E1 27359.698,E2 27359.698} C_VEL
LIN {X 0,Y 568.145,Z 376.27,A -85,B 0,C 180,E1 27356.671,E2 27356.671} C_VEL
LIN {X 0,Y 568.206,Z 376.27,A -85,B 0,C 180,E1 27353.433,E2 27353.433} C_VEL
LIN {X 0,Y 568.143,Z 376.271,A -85,B 0,C 180,E1 27350.376,E2 27350.376} C_VEL
LIN {X 0,Y 568.206,Z 376.257,A -85,B 0,C 180,E1 27347.19,E2 27347.19} C_VEL
LIN {X 0,Y 568.141,Z 376.271,A -85,B 0,C 180,E1 27344.171,E2 27344.171} C_VEL
LIN {X 0,Y 568.212,Z 376.258,A -85,B 0,C 180,E1 27341.002,E2 27341.002} C_VEL
LIN {X 0,Y 568.14,Z 376.272,A -85,B 0,C 180,E1 27337.876,E2 27337.876} C_VEL
LIN {X 0,Y 568.205,Z 376.259,A -85,B 0,C 180,E1 27334.685,E2 27334.685} C_VEL
LIN {X 0,Y 568.139,Z 376.273,A -85,B 0,C 180,E1 27331.63,E2 27331.63} C_VEL
LIN {X 0,Y 568.213,Z 376.261,A -85,B 0,C 180,E1 27328.492,E2 27328.492} C_VEL
LIN {X 0,Y 568.136,Z 376.267,A -85,B 0,C 180,E1 27325.359,E2 27325.359} C_VEL
LIN {X 0,Y 568.213,Z 376.268,A -85,B 0,C 180,E1 27322.194,E2 27322.194} C_VEL
LIN {X 0,Y 568.135,Z 376.277,A -85,B 0,C 180,E1 27319.105,E2 27319.105} C_VEL
LIN {X 0,Y 568.205,Z 376.264,A -85,B 0,C 180,E1 27315.886,E2 27315.886} C_VEL
LIN {X 0,Y 568.223,Z 376.699,A -85,B 0,C 180,E1 27315.493,E2 27315.493} C_VEL
LIN {X 0,Y 569.631,Z 380.025,A -85,B 0,C 180,E1 27315.121,E2 27315.121} C_VEL
LIN {X 0,Y 570.779,Z 381.739,A -85,B 0,C 180,E1 27314.907,E2 27314.907} C_VEL
LIN {X 0,Y 576.774,Z 392.987,A -85,B 0,C 180,E1 27313.688,E2 27313.688} C_VEL
LIN {X 0,Y 575.653,Z 449.741,A -85,B 0,C 180,E1 27310.709,E2 27310.709} C_VEL
LIN {X 0,Y 575.545,Z 466.387,A -85,B 0,C 180,E1 27309.879,E2 27309.879} C_VEL
LIN {X 0,Y 576.445,Z 474.269,A -85,B 0,C 180,E1 27309.679,E2 27309.679} C_VEL
LIN {X 0,Y 575.223,Z 678.909,A -85,B 0,C 180,E1 27306.596,E2 27306.596} C_VEL
LIN {X 0,Y 574.407,Z 815.863,A -85,B 0,C 180,E1 27304.56,E2 27304.56} C_VEL
LIN {X 0,Y 573.996,Z 839.617,A -85,B 0,C 180,E1 27304.021,E2 27304.021} C_VEL
LIN {X 0,Y 573.621,Z 861.177,A -85,B 0,C 180,E1 27303.348,E2 27303.348} C_VEL
LIN {X 0,Y 573.022,Z 883.678,A -85,B 0,C 180,E1 27302.45,E2 27302.45} C_VEL
LIN {X 0,Y 572.504,Z 904.781,A -85,B 0,C 180,E1 27301.421,E2 27301.421} C_VEL
LIN {X 0,Y 571.825,Z 925.929,A -85,B 0,C 180,E1 27300.179,E2 27300.179} C_VEL
LIN {X 0,Y 571.198,Z 947.111,A -85,B 0,C 180,E1 27298.721,E2 27298.721} C_VEL
LIN {X 0,Y 570.577,Z 965.908,A -85,B 0,C 180,E1 27297.218,E2 27297.218} C_VEL
LIN {X 0,Y 570.011,Z 984.455,A -85,B 0,C 180,E1 27295.508,E2 27295.508} C_VEL
LIN {X 0,Y 569.52,Z 1001.615,A -85,B 0,C 180,E1 27293.706,E2 27293.706} C_VEL
LIN {X 0,Y 569.064,Z 1017.692,A -85,B 0,C 180,E1 27291.761,E2 27291.761} C_VEL
LIN {X 0,Y 568.711,Z 1032.333,A -85,B 0,C 180,E1 27289.728,E2 27289.728} C_VEL
LIN {X 0,Y 568.446,Z 1045.008,A -85,B 0,C 180,E1 27287.716,E2 27287.716} C_VEL
LIN {X 0,Y 568.221,Z 1056.317,A -85,B 0,C 180,E1 27285.618,E2 27285.618} C_VEL
LIN {X 0,Y 568.078,Z 1065.996,A -85,B 0,C 180,E1 27283.538,E2 27283.538} C_VEL
LIN {X 0,Y 567.988,Z 1074.477,A -85,B 0,C 180,E1 27281.331,E2 27281.331} C_VEL
LIN {X 0,Y 567.947,Z 1081.172,A -85,B 0,C 180,E1 27279.219,E2 27279.219} C_VEL
LIN {X 0,Y 567.895,Z 1086.634,A -85,B 0,C 180,E1 27276.978,E2 27276.978} C_VEL
LIN {X 0,Y 567.908,Z 1090.276,A -85,B 0,C 180,E1 27274.949,E2 27274.949} C_VEL
LIN {X 0,Y 567.914,Z 1092.988,A -85,B 0,C 180,E1 27272.523,E2 27272.523} C_VEL
LIN {X 0,Y 567.887,Z 1093.917,A -85,B 0,C 180,E1 27270.404,E2 27270.404} C_VEL
LIN {X 0,Y 567.912,Z 1093.323,A -85,B 0,C 180,E1 27267.982,E2 27267.982} C_VEL
LIN {X 0,Y 567.914,Z 1091.276,A -85,B 0,C 180,E1 27265.759,E2 27265.759} C_VEL
LIN {X 0,Y 567.918,Z 1087.46,A -85,B 0,C 180,E1 27263.429,E2 27263.429} C_VEL
LIN {X 0,Y 567.943,Z 1082.55,A -85,B 0,C 180,E1 27261.292,E2 27261.292} C_VEL
LIN {X 0,Y 567.977,Z 1075.763,A -85,B 0,C 180,E1 27259.04,E2 27259.04} C_VEL
LIN {X 0,Y 568.066,Z 1068.107,A -85,B 0,C 180,E1 27256.98,E2 27256.98} C_VEL
LIN {X 0,Y 568.212,Z 1057.61,A -85,B 0,C 180,E1 27254.641,E2 27254.641} C_VEL
LIN {X 0,Y 568.428,Z 1046.236,A -85,B 0,C 180,E1 27252.495,E2 27252.495} C_VEL
LIN {X 0,Y 568.691,Z 1033.042,A -85,B 0,C 180,E1 27250.378,E2 27250.378} C_VEL
LIN {X 0,Y 569.048,Z 1018.537,A -85,B 0,C 180,E1 27248.347,E2 27248.347} C_VEL
LIN {X 0,Y 569.454,Z 1003.475,A -85,B 0,C 180,E1 27246.511,E2 27246.511} C_VEL
LIN {X 0,Y 569.95,Z 986.114,A -85,B 0,C 180,E1 27244.656,E2 27244.656} C_VEL
LIN {X 0,Y 570.535,Z 967.89,A -85,B 0,C 180,E1 27242.949,E2 27242.949} C_VEL
LIN {X 0,Y 571.145,Z 948.606,A -85,B 0,C 180,E1 27241.393,E2 27241.393} C_VEL
LIN {X 0,Y 571.764,Z 927.708,A -85,B 0,C 180,E1 27239.933,E2 27239.933} C_VEL
LIN {X 0,Y 572.4,Z 907.826,A -85,B 0,C 180,E1 27238.748,E2 27238.748} C_VEL
LIN {X 0,Y 572.972,Z 885.415,A -85,B 0,C 180,E1 27237.628,E2 27237.628} C_VEL
LIN {X 0,Y 573.584,Z 863.358,A -85,B 0,C 180,E1 27236.727,E2 27236.727} C_VEL
LIN {X 0,Y 573.98,Z 840.955,A -85,B 0,C 180,E1 27236.017,E2 27236.017} C_VEL
LIN {X 0,Y 574.392,Z 818.109,A -85,B 0,C 180,E1 27235.478,E2 27235.478} C_VEL
LIN {X 0,Y 574.74,Z 764.411,A -85,B 0,C 180,E1 27234.662,E2 27234.662} C_VEL
LIN {X 0,Y 575.912,Z 558.055,A -85,B 0,C 180,E1 27231.595,E2 27231.595} C_VEL
LIN {X 0,Y 576.281,Z 471.463,A -85,B 0,C 180,E1 27230.263,E2 27230.263} C_VEL
LIN {X 0,Y 575.418,Z 464.637,A -85,B 0,C 180,E1 27230.055,E2 27230.055} C_VEL
LIN {X 0,Y 576.503,Z 406.466,A -85,B 0,C 180,E1 27227.031,E2 27227.031} C_VEL
LIN {X 0,Y 576.719,Z 392.842,A -85,B 0,C 180,E1 27226.298,E2 27226.298} C_VEL
LIN {X 0,Y 572.485,Z 384.935,A -85,B 0,C 180,E1 27225.445,E2 27225.445} C_VEL
LIN {X 0,Y 570.153,Z 380.669,A -85,B 0,C 180,E1 27224.969,E2 27224.969} C_VEL
LIN {X 0,Y 568.343,Z 377.284,A -85,B 0,C 180,E1 27224.582,E2 27224.582} C_VEL
LIN {X 0,Y 568.177,Z 376.335,A -85,B 0,C 180,E1 27224.4,E2 27224.4} C_VEL
LIN {X 0,Y 568.14,Z 376.277,A -85,B 0,C 180,E1 27221.129,E2 27221.129} C_VEL
LIN {X 0,Y 568.154,Z 376.268,A -85,B 0,C 180,E1 27218.276,E2 27218.276} C_VEL
LIN {X 0,Y 568.143,Z 376.267,A -85,B 0,C 180,E1 27214.905,E2 27214.905} C_VEL
LIN {X 0,Y 568.159,Z 376.274,A -85,B 0,C 180,E1 27211.979,E2 27211.979} C_VEL
LIN {X 0,Y 568.15,Z 376.273,A -85,B 0,C 180,E1 27208.714,E2 27208.714} C_VEL
LIN {X 0,Y 568.146,Z 376.266,A -85,B 0,C 180,E1 27205.877,E2 27205.877} C_VEL
LIN {X 0,Y 568.153,Z 376.272,A -85,B 0,C 180,E1 27202.45,E2 27202.45} C_VEL
LIN {X 0,Y 568.144,Z 376.262,A -85,B 0,C 180,E1 27199.641,E2 27199.641} C_VEL
LIN {X 0,Y 568.159,Z 376.271,A -85,B 0,C 180,E1 27196.249,E2 27196.249} C_VEL
LIN {X 0,Y 568.143,Z 376.262,A -85,B 0,C 180,E1 27193.432,E2 27193.432} C_VEL
LIN {X 0,Y 568.175,Z 376.27,A -85,B 0,C 180,E1 27190.135,E2 27190.135} C_VEL
LIN {X 0,Y 568.143,Z 376.268,A -85,B 0,C 180,E1 27187.178,E2 27187.178} C_VEL
LIN {X 0,Y 568.185,Z 376.268,A -85,B 0,C 180,E1 27183.935,E2 27183.935} C_VEL
LIN {X 0,Y 568.146,Z 376.27,A -85,B 0,C 180,E1 27180.907,E2 27180.907} C_VEL
LIN {X 0,Y 568.188,Z 376.268,A -85,B 0,C 180,E1 27177.68,E2 27177.68} C_VEL
LIN {X 0,Y 568.146,Z 376.272,A -85,B 0,C 180,E1 27174.648,E2 27174.648} C_VEL
LIN {X 0,Y 568.188,Z 376.27,A -85,B 0,C 180,E1 27171.397,E2 27171.397} C_VEL
LIN {X 0,Y 568.145,Z 376.268,A -85,B 0,C 180,E1 27168.426,E2 27168.426} C_VEL
LIN {X 0,Y 568.201,Z 376.268,A -85,B 0,C 180,E1 27165.217,E2 27165.217} C_VEL
LIN {X 0,Y 568.147,Z 376.271,A -85,B 0,C 180,E1 27162.168,E2 27162.168} C_VEL
LIN {X 0,Y 568.152,Z 376.271,A -85,B 0,C 180,E1 27159.938,E2 27159.938} C_VEL
LIN {X 0,Y 567.194,Z 376.397,A -85,B 0,C 180,E1 27159.162,E2 27159.162} C_VEL
LIN {X 0,Y 560.683,Z 377.208,A -85,B 0,C 180,E1 27156.924,E2 27156.924} C_VEL
LIN {X 0,Y 560.219,Z 377.26,A -85,B 0,C 180,E1 27156.413,E2 27156.413} C_VEL
LIN {X 0,Y 560.234,Z 377.259,A -85,B 0,C 180,E1 27153.4,E2 27153.4} C_VEL
LIN {X 0,Y 560.217,Z 377.244,A -85,B 0,C 180,E1 27150.135,E2 27150.135} C_VEL
LIN {X 0,Y 560.233,Z 377.26,A -85,B 0,C 180,E1 27147.142,E2 27147.142} C_VEL
LIN {X 0,Y 560.215,Z 377.249,A -85,B 0,C 180,E1 27143.777,E2 27143.777} C_VEL
LIN {X 0,Y 560.245,Z 377.263,A -85,B 0,C 180,E1 27140.765,E2 27140.765} C_VEL
LIN {X 0,Y 560.215,Z 377.26,A -85,B 0,C 180,E1 27137.434,E2 27137.434} C_VEL
LIN {X 0,Y 560.266,Z 377.247,A -85,B 0,C 180,E1 27134.305,E2 27134.305} C_VEL
LIN {X 0,Y 560.212,Z 377.252,A -85,B 0,C 180,E1 27131.057,E2 27131.057} C_VEL
LIN {X 0,Y 560.284,Z 377.24,A -85,B 0,C 180,E1 27127.872,E2 27127.872} C_VEL
LIN {X 0,Y 560.258,Z 377.519,A -85,B 0,C 180,E1 27127.085,E2 27127.085} C_VEL
LIN {X 0,Y 561.801,Z 381.168,A -85,B 0,C 180,E1 27126.615,E2 27126.615} C_VEL
LIN {X 0,Y 565.942,Z 391.311,A -85,B 0,C 180,E1 27125.466,E2 27125.466} C_VEL
LIN {X 0,Y 566.204,Z 393.549,A -85,B 0,C 180,E1 27125.272,E2 27125.272} C_VEL
LIN {X 0,Y 565.256,Z 426.41,A -85,B 0,C 180,E1 27122.952,E2 27122.952} C_VEL
LIN {X 0,Y 564.484,Z 470.614,A -85,B 0,C 180,E1 27119.978,E2 27119.978} C_VEL
LIN {X 0,Y 565.695,Z 479.325,A -85,B 0,C 180,E1 27119.778,E2 27119.778} C_VEL
LIN {X 0,Y 564.416,Z 731.793,A -85,B 0,C 180,E1 27116.258,E2 27116.258} C_VEL
LIN {X 0,Y 564.112,Z 752.059,A -85,B 0,C 180,E1 27115.794,E2 27115.794} C_VEL
LIN {X 0,Y 563.721,Z 772.333,A -85,B 0,C 180,E1 27115.138,E2 27115.138} C_VEL
LIN {X 0,Y 563.301,Z 791.697,A -85,B 0,C 180,E1 27114.318,E2 27114.318} C_VEL
LIN {X 0,Y 562.829,Z 810.309,A -85,B 0,C 180,E1 27113.338,E2 27113.338} C_VEL
LIN {X 0,Y 562.317,Z 828.906,A -85,B 0,C 180,E1 27112.146,E2 27112.146} C_VEL
LIN {X 0,Y 561.806,Z 846.375,A -85,B 0,C 180,E1 27110.797,E2 27110.797} C_VEL
LIN {X 0,Y 561.356,Z 862.251,A -85,B 0,C 180,E1 27109.347,E2 27109.347} C_VEL
LIN {X 0,Y 560.957,Z 877.204,A -85,B 0,C 180,E1 27107.746,E2 27107.746} C_VEL
LIN {X 0,Y 560.612,Z 891.149,A -85,B 0,C 180,E1 27105.989,E2 27105.989} C_VEL
LIN {X 0,Y 560.35,Z 903.467,A -85,B 0,C 180,E1 27104.15,E2 27104.15} C_VEL
LIN {X 0,Y 560.17,Z 914.071,A -85,B 0,C 180,E1 27102.263,E2 27102.263} C_VEL
